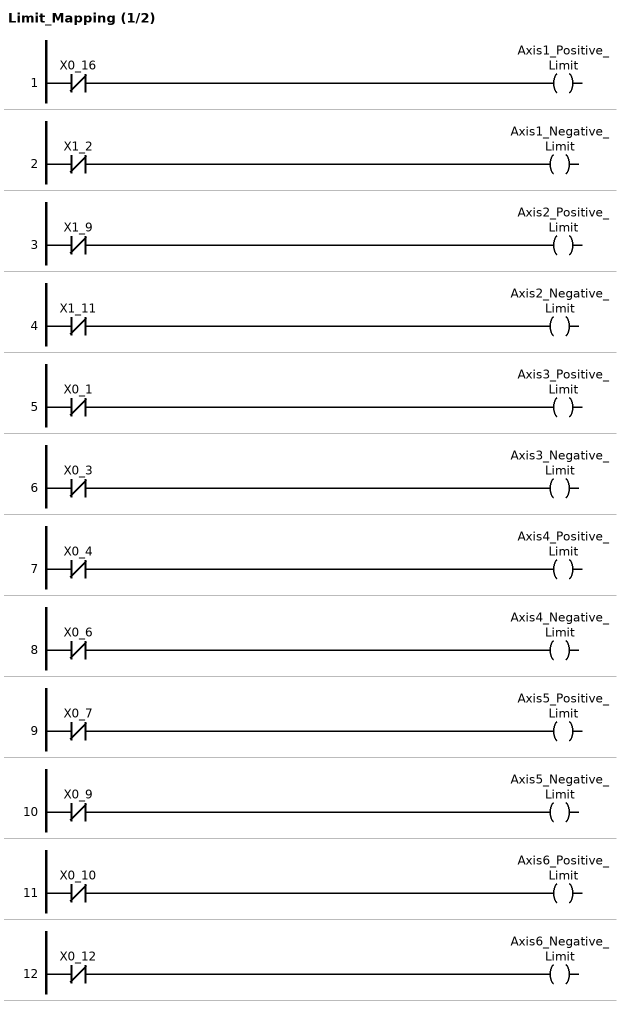
[picture p48: Limit_Mapping (LD)]
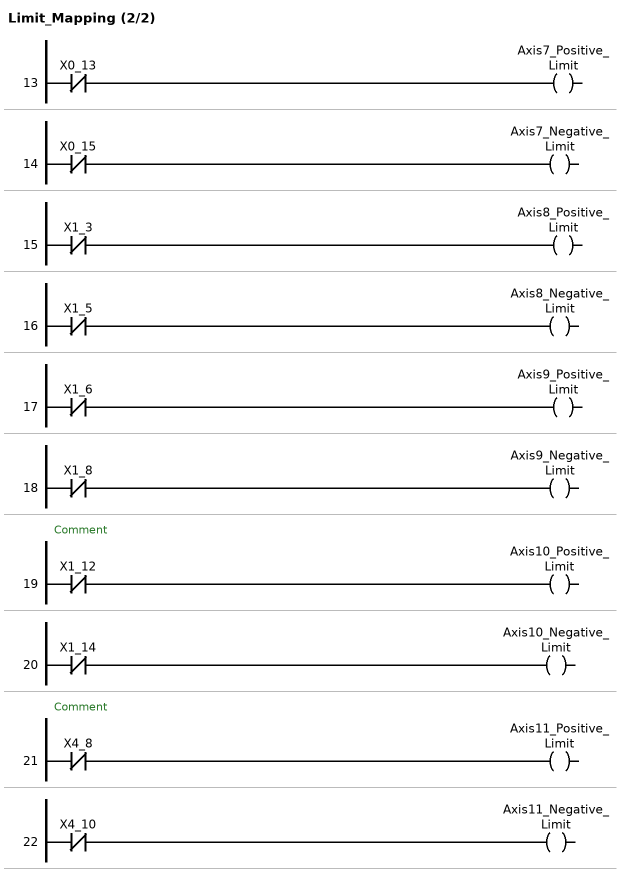
_LD_ (* Ladder Diagram *)
NETWORK 1
	[/X0_16] --- (Axis1_Positive_Limit)
NETWORK 2
	[/X1_2] --- (Axis1_Negative_Limit)
NETWORK 3
	[/X1_9] --- (Axis2_Positive_Limit)
NETWORK 4
	[/X1_11] --- (Axis2_Negative_Limit)
NETWORK 5
	[/X0_1] --- (Axis3_Positive_Limit)
NETWORK 6
	[/X0_3] --- (Axis3_Negative_Limit)
NETWORK 7
	[/X0_4] --- (Axis4_Positive_Limit)
NETWORK 8
	[/X0_6] --- (Axis4_Negative_Limit)
NETWORK 9
	[/X0_7] --- (Axis5_Positive_Limit)
NETWORK 10
	[/X0_9] --- (Axis5_Negative_Limit)
NETWORK 11
	[/X0_10] --- (Axis6_Positive_Limit)
NETWORK 12
	[/X0_12] --- (Axis6_Negative_Limit)
NETWORK 13
	[/X0_13] --- (Axis7_Positive_Limit)
NETWORK 14
	[/X0_15] --- (Axis7_Negative_Limit)
NETWORK 15
	[/X1_3] --- (Axis8_Positive_Limit)
NETWORK 16
	[/X1_5] --- (Axis8_Negative_Limit)
NETWORK 17
	[/X1_6] --- (Axis9_Positive_Limit)
NETWORK 18
	[/X1_8] --- (Axis9_Negative_Limit)
NETWORK 19 (* Comment *)
	[/X1_12] --- (Axis10_Positive_Limit)
NETWORK 20
	[/X1_14] --- (Axis10_Negative_Limit)
NETWORK 21 (* Comment *)
	[/X4_8] --- (Axis11_Positive_Limit)
NETWORK 22
	[/X4_10] --- (Axis11_Negative_Limit)
_END_LD_
(* the same logic as Structured Text *)
(* Network 1 *)
Axis1_Positive_Limit := NOT X0_16;
(* Network 2 *)
Axis1_Negative_Limit := NOT X1_2;
(* Network 3 *)
Axis2_Positive_Limit := NOT X1_9;
(* Network 4 *)
Axis2_Negative_Limit := NOT X1_11;
(* Network 5 *)
Axis3_Positive_Limit := NOT X0_1;
(* Network 6 *)
Axis3_Negative_Limit := NOT X0_3;
(* Network 7 *)
Axis4_Positive_Limit := NOT X0_4;
(* Network 8 *)
Axis4_Negative_Limit := NOT X0_6;
(* Network 9 *)
Axis5_Positive_Limit := NOT X0_7;
(* Network 10 *)
Axis5_Negative_Limit := NOT X0_9;
(* Network 11 *)
Axis6_Positive_Limit := NOT X0_10;
(* Network 12 *)
Axis6_Negative_Limit := NOT X0_12;
(* Network 13 *)
Axis7_Positive_Limit := NOT X0_13;
(* Network 14 *)
Axis7_Negative_Limit := NOT X0_15;
(* Network 15 *)
Axis8_Positive_Limit := NOT X1_3;
(* Network 16 *)
Axis8_Negative_Limit := NOT X1_5;
(* Network 17 *)
Axis9_Positive_Limit := NOT X1_6;
(* Network 18 *)
Axis9_Negative_Limit := NOT X1_8;
(* Network 19: Comment *)
Axis10_Positive_Limit := NOT X1_12;
(* Network 20 *)
Axis10_Negative_Limit := NOT X1_14;
(* Network 21: Comment *)
Axis11_Positive_Limit := NOT X4_8;
(* Network 22 *)
Axis11_Negative_Limit := NOT X4_10;
END_PROGRAM

(* POU Other_Folder/Speed_AxisStatus_IO/Speed_Setting, ST *)
PROGRAM Speed_Setting
VAR
	UP1: R_TRIG;
	UP2: R_TRIG;
	UP3: R_TRIG;

	step: INT;
END_VAR
CASE step OF
0:
step:=1;


1:
UP1(CLK:=M100 , Q=> );
UP2(CLK:=M101 , Q=> );
UP3(CLK:=M102 , Q=> );
(*调速选择*)
IF UP1.Q THEN(*低速*)
D11:=D100[0];D12:=D100[1];D13:=D100[2];D14:=D100[3];D15:=D100[4];
D16:=D100[5];D17:=D100[6];D18:=D100[7];D19:=D100[8];D20:=D100[9];D2_1:=D100[10];D2_2:=D100[11];
step:=10;
END_IF
IF UP2.Q THEN(*中速*)
D11:=D101[0];D12:=D101[1];D13:=D101[2];D14:=D101[3];D15:=D101[4];
D16:=D101[5];D17:=D101[6];D18:=D101[7];D19:=D101[8];D20:=D101[9];D2_1:=D101[10];D2_2:=D101[11];
step:=20;
END_IF
IF UP3.Q THEN(*高速*)
D11:=D102[0];D12:=D102[1];D13:=D102[2];D14:=D102[3];D15:=D102[4];
D16:=D102[5];D17:=D102[6];D18:=D102[7];D19:=D102[8];D20:=D102[9];D2_1:=D102[10];D2_2:=D102[11];
step:=30;
END_IF

10:
M101:=FALSE;
M102:=FALSE;
step:=1;

20:
M100:=FALSE;
M102:=FALSE;
step:=1;

30:
M100:=FALSE;
M101:=FALSE;
step:=1;


END_CASE
END_PROGRAM

(* POU Debug_Folder/Axis1_Debug_Model, ST *)
PROGRAM Axis1_Debug_Model
VAR
	UP1: R_TRIG;
	UP2: R_TRIG;
	UP3: R_TRIG;
	UP4: R_TRIG;
	step:INT;
END_VAR
UP1(CLK:=Axis1_debug_trigger , Q=> );

CASE step OF
0:
IF UP1.Q THEN
step:=1;
END_IF;

1:
(*点动加-----------
点动减------------
手动点动-----------*)
UP2(CLK:=Axis1_mov_add , Q=> );
UP3(CLK:=Axis1_mov_sub , Q=> );
UP4(CLK:=Axis1_mov_line , Q=> );

IF UP2.Q AND Debug_Model AND Axis1_Poweron AND NOT Total_Pause THEN
D1:=Axis1.NcToPlc.ActPos+D200;
Axis1_mov_add:=FALSE;
step:=10;
ELSE
Axis1_mov_add:=FALSE;
Axis1_MoveAbsolute:=FALSE;
END_IF

IF UP3.Q AND Debug_Model AND Axis1_Poweron AND NOT Total_Pause THEN
D1:=Axis1.NcToPlc.ActPos-D200;
Axis1_mov_sub:=FALSE;
step:=10;
ELSE
Axis1_mov_sub:=FALSE;
Axis1_MoveAbsolute:=FALSE;
END_IF

IF UP4.Q AND Debug_Model AND Axis1_Poweron  AND NOT Total_Pause THEN
D1:=D201;
Axis1_mov_line:=FALSE;
step:=10;
ELSE
Axis1_mov_line:=FALSE;
Axis1_MoveAbsolute:=FALSE;
END_IF

10:
Axis1_MoveAbsolute:=TRUE;
IF Axis1_Abs_Function.Done THEN
Axis1_MoveAbsolute:=FALSE;
step:=1;
END_IF

END_CASE

IF Axis1_mov_add THEN
Axis1_mov_add:=FALSE;
END_IF
IF Axis1_mov_sub THEN
Axis1_mov_sub:=FALSE;
END_IF
IF Axis1_mov_line THEN
Axis1_mov_line:=FALSE;
END_IF


IF NOT Debug_Model  THEN
Axis1_debug_trigger:=FALSE;
step:=0;
END_IF

IF Total_Emergency THEN
Axis1_debug_trigger:=FALSE;
Axis1_mov_add:=FALSE;
Axis1_mov_sub:=FALSE;
Axis1_mov_line:=FALSE;
Axis1_MoveAbsolute:=FALSE;
step:=0;
END_IF
END_PROGRAM

(* POU Debug_Folder/Axis2_Debug_Model, ST *)
PROGRAM Axis2_Debug_Model
VAR
	UP1: R_TRIG;
	UP2: R_TRIG;
	UP3: R_TRIG;
	UP4: R_TRIG;
	step:INT;

END_VAR
UP1(CLK:=Axis2_debug_trigger , Q=> );

CASE step OF
0:
IF UP1.Q THEN
step:=1;
END_IF;

1:
UP2(CLK:=Axis2_mov_add , Q=> );
UP3(CLK:=Axis2_mov_sub , Q=> );
UP4(CLK:=Axis2_mov_line , Q=> );

IF UP2.Q AND Debug_Model AND Axis2_Poweron AND NOT Total_Pause THEN
D2:=Axis2.NcToPlc.ActPos+D200;
Axis2_mov_add:=FALSE;
step:=10;
ELSE
Axis2_mov_add:=FALSE;
Axis2_MoveAbsolute:=FALSE;
END_IF

IF UP3.Q AND Debug_Model AND Axis2_Poweron AND NOT Total_Pause THEN
D2:=Axis2.NcToPlc.ActPos-D200;
Axis2_mov_sub:=FALSE;
step:=10;
ELSE
Axis2_mov_sub:=FALSE;
Axis2_MoveAbsolute:=FALSE;
END_IF

IF UP4.Q AND Debug_Model AND Axis2_Poweron AND NOT Total_Pause THEN
D2:=D202;
Axis2_mov_line:=FALSE;
step:=10;
ELSE
Axis2_mov_line:=FALSE;
Axis2_MoveAbsolute:=FALSE;
END_IF

10:
Axis2_MoveAbsolute:=TRUE;
IF Axis2_Abs_Function.Done THEN
Axis2_MoveAbsolute:=FALSE;
step:=1;
END_IF

END_CASE

IF Axis2_mov_add THEN
Axis2_mov_add:=FALSE;
END_IF
IF Axis2_mov_sub THEN
Axis2_mov_sub:=FALSE;
END_IF
IF Axis2_mov_line THEN
Axis2_mov_line:=FALSE;
END_IF


IF NOT Debug_Model  THEN
Axis2_debug_trigger:=FALSE;
step:=0;
END_IF

IF Total_Emergency THEN
Axis2_debug_trigger:=FALSE;
Axis2_mov_add:=FALSE;
Axis2_mov_sub:=FALSE;
Axis2_mov_line:=FALSE;
Axis2_MoveAbsolute:=FALSE;
step:=0;
END_IF
END_PROGRAM

(* POU Debug_Folder/Axis3_Debug_Model, ST *)
PROGRAM Axis3_Debug_Model
VAR
	UP1: R_TRIG;
	UP2: R_TRIG;
	UP3: R_TRIG;
	UP4: R_TRIG;
	step:INT;
END_VAR
UP1(CLK:=Axis3_debug_trigger , Q=> );

CASE step OF
0:
IF UP1.Q THEN
step:=1;
END_IF;

1:
UP2(CLK:=Axis3_mov_add , Q=> );
UP3(CLK:=Axis3_mov_sub , Q=> );
UP4(CLK:=Axis3_mov_line , Q=> );

IF UP2.Q AND Debug_Model AND Axis3_Poweron AND NOT Total_Pause THEN
D3:=Axis3.NcToPlc.ActPos+D200;
Axis3_mov_add:=FALSE;
step:=10;
ELSE
Axis3_mov_add:=FALSE;
Axis3_MoveAbsolute:=FALSE;
END_IF

IF UP3.Q AND Debug_Model AND Axis3_Poweron AND NOT Total_Pause THEN
D3:=Axis3.NcToPlc.ActPos-D200;
Axis3_mov_sub:=FALSE;
step:=10;
ELSE
Axis3_mov_sub:=FALSE;
Axis3_MoveAbsolute:=FALSE;
END_IF

IF UP4.Q AND Debug_Model AND Axis3_Poweron AND NOT Total_Pause THEN
D3:=D203;
Axis3_mov_line:=FALSE;
step:=10;
ELSE
Axis3_mov_line:=FALSE;
Axis3_MoveAbsolute:=FALSE;
END_IF

10:
Axis3_MoveAbsolute:=TRUE;
IF Axis3_Abs_Function.Done THEN
Axis3_MoveAbsolute:=FALSE;
step:=1;
END_IF

END_CASE

IF Axis3_mov_add THEN
Axis3_mov_add:=FALSE;
END_IF
IF Axis3_mov_sub THEN
Axis3_mov_sub:=FALSE;
END_IF
IF Axis3_mov_line THEN
Axis3_mov_line:=FALSE;
END_IF


IF NOT Debug_Model  THEN
Axis3_debug_trigger:=FALSE;
step:=0;
END_IF

IF Total_Emergency THEN
Axis3_debug_trigger:=FALSE;
Axis3_mov_add:=FALSE;
Axis3_mov_sub:=FALSE;
Axis3_mov_line:=FALSE;
Axis3_MoveAbsolute:=FALSE;
step:=0;
END_IF
END_PROGRAM

(* POU Debug_Folder/Axis4_Debug_Model, ST *)
PROGRAM Axis4_Debug_Model
VAR
	UP1: R_TRIG;
	UP2: R_TRIG;
	UP3: R_TRIG;
	UP4: R_TRIG;
	step:INT;
	M1:BOOL;


END_VAR
UP1(CLK:=Axis4_debug_trigger , Q=> );

CASE step OF
0:
IF UP1.Q THEN
step:=1;
END_IF;

1:
UP2(CLK:=Axis4_mov_add , Q=> );
IF UP2.Q AND Debug_Model AND Axis4_Poweron  AND NOT Total_Pause THEN
D4:=Axis4.NcToPlc.ActPos+D200;
Axis4_mov_add:=FALSE;
step:=10;
ELSE
Axis4_mov_add:=FALSE;
Axis4_MoveAbsolute:=FALSE;
END_IF


UP3(CLK:=Axis4_mov_sub , Q=> );
IF UP3.Q AND Debug_Model AND Axis4_Poweron  AND NOT Total_Pause  THEN
D4:=Axis4.NcToPlc.ActPos-D200;
Axis4_mov_sub:=FALSE;
step:=10;
ELSE
Axis4_mov_sub:=FALSE;
Axis4_MoveAbsolute:=FALSE;
END_IF


UP4(CLK:=Axis4_mov_line , Q=> );
IF UP4.Q AND Debug_Model AND Axis4_Poweron  AND NOT Total_Pause  THEN
D4:=D204;
Axis4_mov_line:=FALSE;
step:=10;
ELSE
Axis4_mov_line:=FALSE;
Axis4_MoveAbsolute:=FALSE;
END_IF


10:
Axis4_MoveAbsolute:=TRUE;
IF Axis4_Abs_Function.Done THEN
Axis4_MoveAbsolute:=FALSE;
step:=1;
END_IF


END_CASE

IF Axis4_mov_add THEN
Axis4_mov_add:=FALSE;
END_IF
IF Axis4_mov_sub THEN
Axis4_mov_sub:=FALSE;
END_IF
IF Axis4_mov_line THEN
Axis4_mov_line:=FALSE;
END_IF


IF NOT Debug_Model  THEN
Axis4_debug_trigger:=FALSE;
step:=0;
END_IF

IF Total_Emergency THEN
Axis4_debug_trigger:=FALSE;
Axis4_mov_add:=FALSE;
Axis4_mov_sub:=FALSE;
Axis4_mov_line:=FALSE;
Axis4_MoveAbsolute:=FALSE;
Axis4_1_MoveAbsolute:=FALSE;
step:=0;
END_IF
END_PROGRAM

(* POU Debug_Folder/Axis5_Debug_Model, ST *)
PROGRAM Axis5_Debug_Model
VAR
	UP1: R_TRIG;
	UP2: R_TRIG;
	UP3: R_TRIG;
	UP4: R_TRIG;
	step:INT;
END_VAR
UP1(CLK:=Axis5_debug_trigger , Q=> );

CASE step OF
0:
IF UP1.Q THEN
step:=1;
END_IF;

1:
UP2(CLK:=Axis5_mov_add , Q=> );
UP3(CLK:=Axis5_mov_sub , Q=> );
UP4(CLK:=Axis5_mov_line , Q=> );

IF UP2.Q AND Debug_Model AND Axis5_Poweron  AND NOT Total_Pause THEN
D5:=Axis5.NcToPlc.ActPos+D200;
Axis5_mov_add:=FALSE;
step:=10;
ELSE
Axis5_mov_add:=FALSE;
Axis5_MoveAbsolute:=FALSE;
END_IF

IF UP3.Q AND Debug_Model AND Axis5_Poweron AND NOT Total_Pause THEN
D5:=Axis5.NcToPlc.ActPos-D200;
Axis5_mov_sub:=FALSE;
step:=10;
ELSE
Axis5_mov_sub:=FALSE;
Axis5_MoveAbsolute:=FALSE;
END_IF

IF UP4.Q AND Debug_Model AND Axis5_Poweron  AND NOT Total_Pause THEN
D5:=D205;
Axis5_mov_line:=FALSE;
step:=10;
ELSE
Axis5_mov_line:=FALSE;
Axis5_MoveAbsolute:=FALSE;
END_IF

10:
Axis5_MoveAbsolute:=TRUE;
IF Axis5_Abs_Function.Done THEN
Axis5_MoveAbsolute:=FALSE;
step:=1;
END_IF

END_CASE

IF Axis5_mov_add THEN
Axis5_mov_add:=FALSE;
END_IF
IF Axis5_mov_sub THEN
Axis5_mov_sub:=FALSE;
END_IF
IF Axis5_mov_line THEN
Axis5_mov_line:=FALSE;
END_IF


IF NOT Debug_Model  THEN
Axis5_debug_trigger:=FALSE;
step:=0;
END_IF

IF Total_Emergency THEN
Axis5_debug_trigger:=FALSE;
Axis5_mov_add:=FALSE;
Axis5_mov_sub:=FALSE;
Axis5_mov_line:=FALSE;
Axis5_MoveAbsolute:=FALSE;
Axis5_1_MoveAbsolute:=FALSE;
step:=0;
END_IF
END_PROGRAM

(* POU Debug_Folder/Axis6_Debug_Model, ST *)
PROGRAM Axis6_Debug_Model
VAR
	UP1: R_TRIG;
	UP2: R_TRIG;
	UP3: R_TRIG;
	UP4: R_TRIG;
	step:INT;
END_VAR
UP1(CLK:=Axis6_debug_trigger , Q=> );

CASE step OF
0:
IF UP1.Q THEN
step:=1;
END_IF;

1:
UP2(CLK:=Axis6_mov_add , Q=> );
UP3(CLK:=Axis6_mov_sub , Q=> );
UP4(CLK:=Axis6_mov_line , Q=> );

IF UP2.Q AND Debug_Model AND Axis6_Poweron  AND NOT Total_Pause THEN
D6:=Axis6.NcToPlc.ActPos+D200;
Axis6_mov_add:=FALSE;
step:=10;
ELSE
Axis6_mov_add:=FALSE;
Axis6_MoveAbsolute:=FALSE;
END_IF

IF UP3.Q AND Debug_Model AND Axis6_Poweron AND NOT Total_Pause THEN
D6:=Axis6.NcToPlc.ActPos-D200;
Axis6_mov_sub:=FALSE;
step:=10;
ELSE
Axis6_mov_sub:=FALSE;
Axis6_MoveAbsolute:=FALSE;
END_IF

IF UP4.Q AND Debug_Model AND Axis6_Poweron  AND NOT Total_Pause THEN
D6:=D206;
Axis6_mov_line:=FALSE;
step:=10;
ELSE
Axis6_mov_line:=FALSE;
Axis6_MoveAbsolute:=FALSE;
END_IF

10:
Axis6_MoveAbsolute:=TRUE;
IF Axis6_Abs_Function.Done THEN
Axis6_MoveAbsolute:=FALSE;
step:=1;
END_IF
END_CASE

IF Axis6_mov_add THEN
Axis6_mov_add:=FALSE;
END_IF
IF Axis6_mov_sub THEN
Axis6_mov_sub:=FALSE;
END_IF
IF Axis6_mov_line THEN
Axis6_mov_line:=FALSE;
END_IF


IF NOT Debug_Model  THEN
Axis6_debug_trigger:=FALSE;
step:=0;
END_IF

IF Total_Emergency THEN
Axis6_debug_trigger:=FALSE;
Axis6_mov_add:=FALSE;
Axis6_mov_sub:=FALSE;
Axis6_mov_line:=FALSE;
Axis6_MoveAbsolute:=FALSE;
step:=0;
END_IF
END_PROGRAM

(* POU Debug_Folder/Axis7_Debug_Model, ST *)
PROGRAM Axis7_Debug_Model
VAR
	UP1: R_TRIG;
	UP2: R_TRIG;
	UP3: R_TRIG;
	UP4: R_TRIG;
	step:INT;
END_VAR
UP1(CLK:=Axis7_debug_trigger , Q=> );

CASE step OF
0:
IF UP1.Q THEN
step:=1;
END_IF;

1:
UP2(CLK:=Axis7_mov_add , Q=> );
UP3(CLK:=Axis7_mov_sub , Q=> );
UP4(CLK:=Axis7_mov_line , Q=> );

IF UP2.Q AND Debug_Model AND Axis7_Poweron  AND NOT Total_Pause THEN
D7:=Axis7.NcToPlc.ActPos+D200;
Axis7_mov_add:=FALSE;
step:=10;
ELSE
Axis7_mov_add:=FALSE;
Axis7_MoveAbsolute:=FALSE;
END_IF

IF UP3.Q AND Debug_Model AND Axis7_Poweron AND NOT Total_Pause THEN
D7:=Axis7.NcToPlc.ActPos-D200;
Axis7_mov_sub:=FALSE;
step:=10;
ELSE
Axis7_mov_sub:=FALSE;
Axis7_MoveAbsolute:=FALSE;
END_IF

IF UP4.Q AND Debug_Model AND Axis7_Poweron  AND NOT Total_Pause THEN
D7:=D207;
Axis7_mov_line:=FALSE;
step:=10;
ELSE
Axis7_mov_line:=FALSE;
Axis7_MoveAbsolute:=FALSE;
END_IF

10:
Axis7_MoveAbsolute:=TRUE;
IF Axis7_Abs_Function.Done THEN
Axis7_MoveAbsolute:=FALSE;
step:=1;
END_IF
END_CASE

IF Axis7_mov_add THEN
Axis7_mov_add:=FALSE;
END_IF
IF Axis7_mov_sub THEN
Axis7_mov_sub:=FALSE;
END_IF
IF Axis7_mov_line THEN
Axis7_mov_line:=FALSE;
END_IF


IF NOT Debug_Model  THEN
Axis7_debug_trigger:=FALSE;
step:=0;
END_IF

IF Total_Emergency THEN
Axis7_debug_trigger:=FALSE;
Axis7_mov_add:=FALSE;
Axis7_mov_sub:=FALSE;
Axis7_mov_line:=FALSE;
Axis7_MoveAbsolute:=FALSE;
step:=0;
END_IF
END_PROGRAM

(* POU Debug_Folder/Axis8_Debug_Model, ST *)
PROGRAM Axis8_Debug_Model
VAR
	UP1: R_TRIG;
	UP2: R_TRIG;
	UP3: R_TRIG;
	UP4: R_TRIG;
	step:INT;
END_VAR
UP1(CLK:=Axis8_debug_trigger , Q=> );

CASE step OF
0:
IF UP1.Q THEN
step:=1;
END_IF;

1:
UP2(CLK:=Axis8_mov_add , Q=> );
UP3(CLK:=Axis8_mov_sub , Q=> );
UP4(CLK:=Axis8_mov_line , Q=> );

IF UP2.Q AND Debug_Model AND Axis8_Poweron  AND NOT Total_Pause THEN
D8:=Axis8.NcToPlc.ActPos+D200;
Axis8_mov_add:=FALSE;
step:=10;
ELSE
Axis8_mov_add:=FALSE;
Axis8_MoveAbsolute:=FALSE;
END_IF

IF UP3.Q AND Debug_Model AND Axis8_Poweron AND NOT Total_Pause THEN
D8:=Axis8.NcToPlc.ActPos-D200;
Axis8_mov_sub:=FALSE;
step:=10;
ELSE
Axis8_mov_sub:=FALSE;
Axis8_MoveAbsolute:=FALSE;
END_IF

IF UP4.Q AND Debug_Model AND Axis8_Poweron  AND NOT Total_Pause THEN
D8:=D208;
Axis8_mov_line:=FALSE;
step:=10;
ELSE
Axis8_mov_line:=FALSE;
Axis8_MoveAbsolute:=FALSE;
END_IF

10:
Axis8_MoveAbsolute:=TRUE;
IF Axis8_Abs_Function.Done THEN
Axis8_MoveAbsolute:=FALSE;
step:=1;
END_IF
END_CASE

IF Axis8_mov_add THEN
Axis8_mov_add:=FALSE;
END_IF
IF Axis8_mov_sub THEN
Axis8_mov_sub:=FALSE;
END_IF
IF Axis8_mov_line THEN
Axis8_mov_line:=FALSE;
END_IF


IF NOT Debug_Model  THEN
Axis8_debug_trigger:=FALSE;
step:=0;
END_IF

IF Total_Emergency THEN
Axis8_debug_trigger:=FALSE;
Axis8_mov_add:=FALSE;
Axis8_mov_sub:=FALSE;
Axis8_mov_line:=FALSE;
Axis8_MoveAbsolute:=FALSE;
step:=0;
END_IF
END_PROGRAM

(* POU Debug_Folder/Axis9_Debug_Model, ST *)
PROGRAM Axis9_Debug_Model
VAR
	UP1: R_TRIG;
	UP2: R_TRIG;
	UP3: R_TRIG;
	UP4: R_TRIG;
	step:INT;
END_VAR
UP1(CLK:=Axis9_debug_trigger , Q=> );

CASE step OF
0:
IF UP1.Q THEN
step:=1;
END_IF;

1:
UP2(CLK:=Axis9_mov_add , Q=> );
UP3(CLK:=Axis9_mov_sub , Q=> );
UP4(CLK:=Axis9_mov_line , Q=> );

IF UP2.Q AND Debug_Model AND Axis9_Poweron  AND NOT Total_Pause THEN
D9:=Axis9.NcToPlc.ActPos+D200;
Axis9_mov_add:=FALSE;
step:=10;
ELSE
Axis9_mov_add:=FALSE;
Axis9_MoveAbsolute:=FALSE;
END_IF

IF UP3.Q AND Debug_Model AND Axis9_Poweron AND NOT Total_Pause THEN
D9:=Axis9.NcToPlc.ActPos-D200;
Axis9_mov_sub:=FALSE;
step:=10;
ELSE
Axis9_mov_sub:=FALSE;
Axis9_MoveAbsolute:=FALSE;
END_IF

IF UP4.Q AND Debug_Model AND Axis9_Poweron  AND NOT Total_Pause THEN
D9:=D209;
Axis9_mov_line:=FALSE;
step:=10;
ELSE
Axis9_mov_line:=FALSE;
Axis9_MoveAbsolute:=FALSE;
END_IF

10:
Axis9_MoveAbsolute:=TRUE;
IF Axis9_Abs_Function.Done THEN
Axis9_MoveAbsolute:=FALSE;
step:=1;
END_IF
END_CASE

IF Axis9_mov_add THEN
Axis9_mov_add:=FALSE;
END_IF
IF Axis9_mov_sub THEN
Axis9_mov_sub:=FALSE;
END_IF
IF Axis9_mov_line THEN
Axis9_mov_line:=FALSE;
END_IF


IF NOT Debug_Model  THEN
Axis9_debug_trigger:=FALSE;
step:=0;
END_IF

IF Total_Emergency THEN
Axis9_debug_trigger:=FALSE;
Axis9_mov_add:=FALSE;
Axis9_mov_sub:=FALSE;
Axis9_mov_line:=FALSE;
Axis9_MoveAbsolute:=FALSE;
step:=0;
END_IF
END_PROGRAM

(* POU Debug_Folder/Axis10_Debug_Model, ST *)
PROGRAM Axis10_Debug_Model
VAR
	UP1: R_TRIG;
	UP2: R_TRIG;
	UP3: R_TRIG;
	UP4: R_TRIG;
	step:INT;
END_VAR
UP1(CLK:=Axis10_debug_trigger , Q=> );

CASE step OF
0:
IF UP1.Q THEN
step:=1;
END_IF;

1:
UP2(CLK:=Axis10_mov_add , Q=> );
UP3(CLK:=Axis10_mov_sub , Q=> );
UP4(CLK:=Axis10_mov_line , Q=> );

IF UP2.Q AND Debug_Model AND Axis10_Poweron  AND NOT Total_Pause THEN
D10:=Axis10.NcToPlc.ActPos+D200;
Axis10_mov_add:=FALSE;
step:=10;
ELSE
Axis10_mov_add:=FALSE;
Axis10_MoveAbsolute:=FALSE;
END_IF

IF UP3.Q AND Debug_Model AND Axis10_Poweron AND NOT Total_Pause THEN
D10:=Axis10.NcToPlc.ActPos-D200;
Axis10_mov_sub:=FALSE;
step:=10;
ELSE
Axis10_mov_sub:=FALSE;
Axis10_MoveAbsolute:=FALSE;
END_IF

IF UP4.Q AND Debug_Model AND Axis10_Poweron  AND NOT Total_Pause THEN
D10:=D210;
Axis10_mov_line:=FALSE;
step:=10;
ELSE
Axis10_mov_line:=FALSE;
Axis10_MoveAbsolute:=FALSE;
END_IF

10:
Axis10_MoveAbsolute:=TRUE;
IF Axis10_Abs_Function.Done THEN
Axis10_MoveAbsolute:=FALSE;
step:=1;
END_IF
END_CASE

IF Axis10_mov_add THEN
Axis10_mov_add:=FALSE;
END_IF
IF Axis10_mov_sub THEN
Axis10_mov_sub:=FALSE;
END_IF
IF Axis10_mov_line THEN
Axis10_mov_line:=FALSE;
END_IF


IF NOT Debug_Model  THEN
Axis10_debug_trigger:=FALSE;
step:=0;
END_IF

IF Total_Emergency THEN
Axis10_debug_trigger:=FALSE;
Axis10_mov_add:=FALSE;
Axis10_mov_sub:=FALSE;
Axis10_mov_line:=FALSE;
Axis10_MoveAbsolute:=FALSE;
step:=0;
END_IF
END_PROGRAM

(* POU Debug_Folder/Axis11_Debug_Model, ST *)
PROGRAM Axis11_Debug_Model
VAR

	UP1: R_TRIG;
	UP2: R_TRIG;
	UP3: R_TRIG;
	UP4: R_TRIG;
	step:INT;
END_VAR
UP1(CLK:=Axis11_debug_trigger , Q=> );

CASE step OF
0:
IF UP1.Q THEN
step:=1;
END_IF;

1:
UP2(CLK:=Axis11_mov_add , Q=> );
UP3(CLK:=Axis11_mov_sub , Q=> );
UP4(CLK:=Axis11_mov_line , Q=> );

IF UP2.Q AND Debug_Model AND Axis11_Poweron  AND NOT Total_Pause THEN
D1_1:=Axis11.NcToPlc.ActPos+D200;
Axis11_mov_add:=FALSE;
step:=10;
ELSE
Axis11_mov_add:=FALSE;
Axis11_MoveAbsolute:=FALSE;
END_IF

IF UP3.Q AND Debug_Model AND Axis11_Poweron AND NOT Total_Pause THEN
D1_1:=Axis11.NcToPlc.ActPos-D200;
Axis11_mov_sub:=FALSE;
step:=10;
ELSE
Axis11_mov_sub:=FALSE;
Axis11_MoveAbsolute:=FALSE;
END_IF

IF UP4.Q AND Debug_Model AND Axis11_Poweron  AND NOT Total_Pause THEN
D1_1:=D211;
Axis11_mov_line:=FALSE;
step:=10;
ELSE
Axis11_mov_line:=FALSE;
Axis11_MoveAbsolute:=FALSE;
END_IF

10:
Axis11_MoveAbsolute:=TRUE;
IF Axis11_Abs_Function.Done THEN
Axis11_MoveAbsolute:=FALSE;
step:=1;
END_IF
END_CASE

IF Axis11_mov_add THEN
Axis11_mov_add:=FALSE;
END_IF
IF Axis11_mov_sub THEN
Axis11_mov_sub:=FALSE;
END_IF
IF Axis11_mov_line THEN
Axis11_mov_line:=FALSE;
END_IF


IF NOT Debug_Model  THEN
Axis11_debug_trigger:=FALSE;
step:=0;
END_IF

IF Total_Emergency THEN
Axis11_debug_trigger:=FALSE;
Axis11_mov_add:=FALSE;
Axis11_mov_sub:=FALSE;
Axis11_mov_line:=FALSE;
Axis11_MoveAbsolute:=FALSE;
step:=0;
END_IF
END_PROGRAM

(* POU Debug_Folder/Others_Debug_Model, LD *)
PROGRAM Others_Debug_Model
VAR
END_VAR
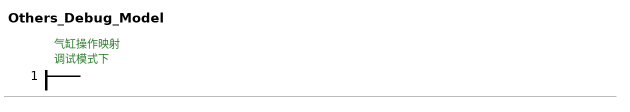
_LD_ (* Ladder Diagram *)
NETWORK 1 (* 气缸操作映射 / 调试模式下 *)
	*
_END_LD_
(* the same logic as Structured Text *)
(* Network 1: 气缸操作映射 / 调试模式下 *)
END_PROGRAM

(* POU Other_Folder/Akam_Stop_Message/Initialization_Folder/Debug12, LD *)
	PROGRAM Debug12
VAR
	t1: TON;
END_VAR
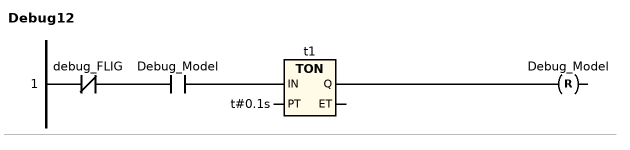
_LD_ (* Ladder Diagram *)
NETWORK 1
	[/debug_FLIG] - [Debug_Model] - t1:TON(IN: *, PT: t#0.1s) --- (R Debug_Model)
_END_LD_
(* the same logic as Structured Text *)
(* Network 1 *)
t1(IN := NOT debug_FLIG AND Debug_Model, PT := t#0.1s);
IF t1.Q THEN Debug_Model := FALSE; END_IF;
END_PROGRAM

(* POU Run_Main_Folder/Feed_alam_status, LD *)
PROGRAM Feed_alam_status
VAR


END_VAR
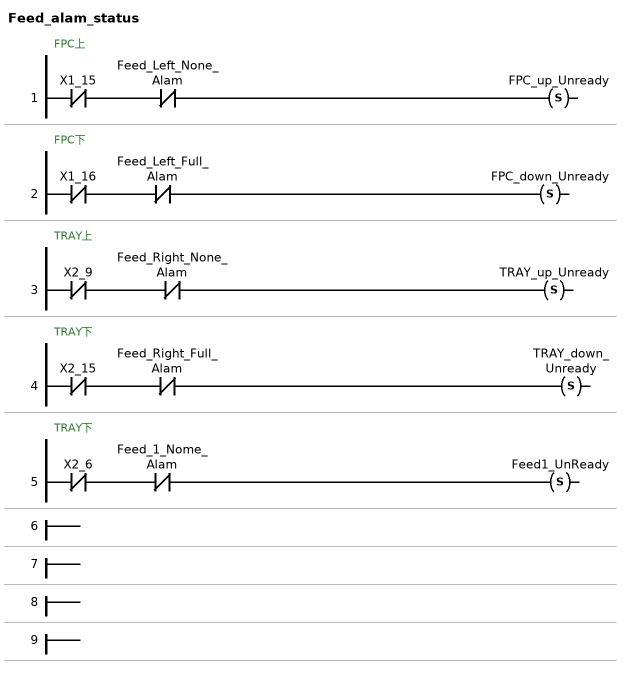
_LD_ (* Ladder Diagram *)
NETWORK 1 (* FPC上 *)
	[/X1_15] - [/Feed_Left_None_Alam] --- (S FPC_up_Unready)
NETWORK 2 (* FPC下 *)
	[/X1_16] - [/Feed_Left_Full_Alam] --- (S FPC_down_Unready)
NETWORK 3 (* TRAY上 *)
	[/X2_9] - [/Feed_Right_None_Alam] --- (S TRAY_up_Unready)
NETWORK 4 (* TRAY下 *)
	[/X2_15] - [/Feed_Right_Full_Alam] --- (S TRAY_down_Unready)
NETWORK 5 (* TRAY下 *)
	[/X2_6] - [/Feed_1_Nome_Alam] --- (S Feed1_UnReady)
NETWORK 6
	*
NETWORK 7
	*
NETWORK 8
	*
NETWORK 9
	*
_END_LD_
(* the same logic as Structured Text *)
(* Network 1: FPC上 *)
IF NOT X1_15 AND NOT Feed_Left_None_Alam THEN FPC_up_Unready := TRUE; END_IF;
(* Network 2: FPC下 *)
IF NOT X1_16 AND NOT Feed_Left_Full_Alam THEN FPC_down_Unready := TRUE; END_IF;
(* Network 3: TRAY上 *)
IF NOT X2_9 AND NOT Feed_Right_None_Alam THEN TRAY_up_Unready := TRUE; END_IF;
(* Network 4: TRAY下 *)
IF NOT X2_15 AND NOT Feed_Right_Full_Alam THEN TRAY_down_Unready := TRUE; END_IF;
(* Network 5: TRAY下 *)
IF NOT X2_6 AND NOT Feed_1_Nome_Alam THEN Feed1_UnReady := TRUE; END_IF;
(* Network 6 *)
(* Network 7 *)
(* Network 8 *)
(* Network 9 *)
END_PROGRAM

(* POU Other_Folder/Home_Back/Axis1_Home_Back, LD *)
PROGRAM Axis1_Home_Back
VAR
	UP1: R_TRIG;
	M1: BOOL;
	M2: BOOL;
	UP2: R_TRIG;
	T1: TON;
	M3: BOOL;
	M4: BOOL;
	DOWN1: F_TRIG;
	M20: BOOL;
END_VAR
VAR (* helpers for the ST form of the networks *)
	_p1 : BOOL;
	_p2 : BOOL;
	_p3 : BOOL;
END_VAR
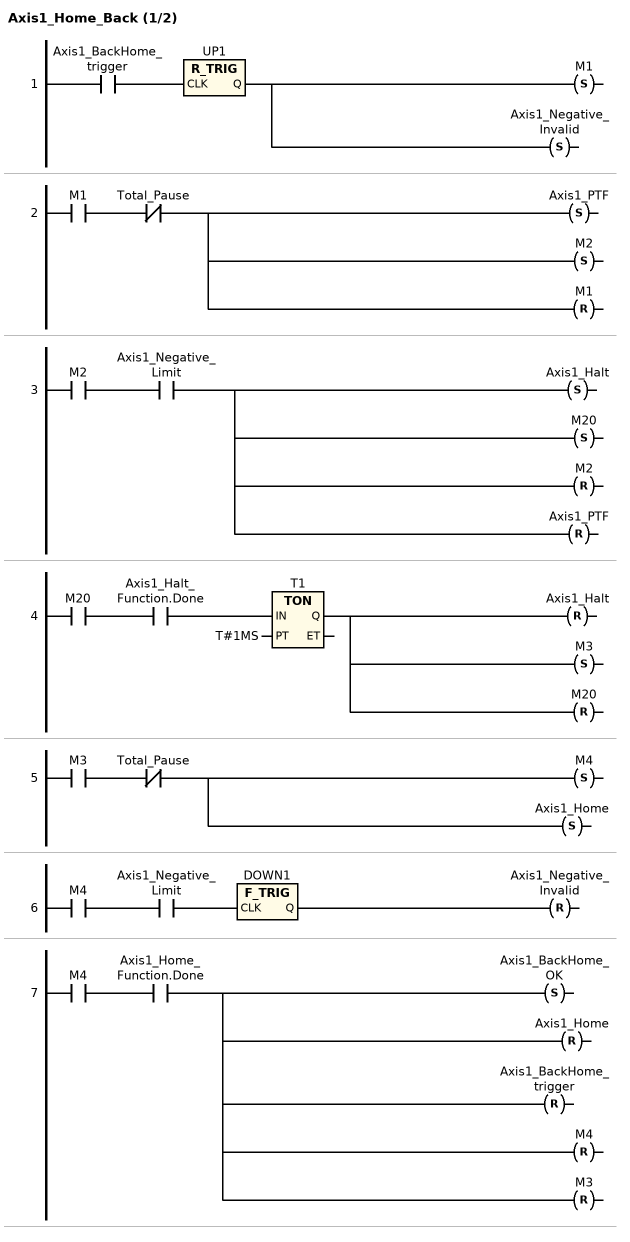
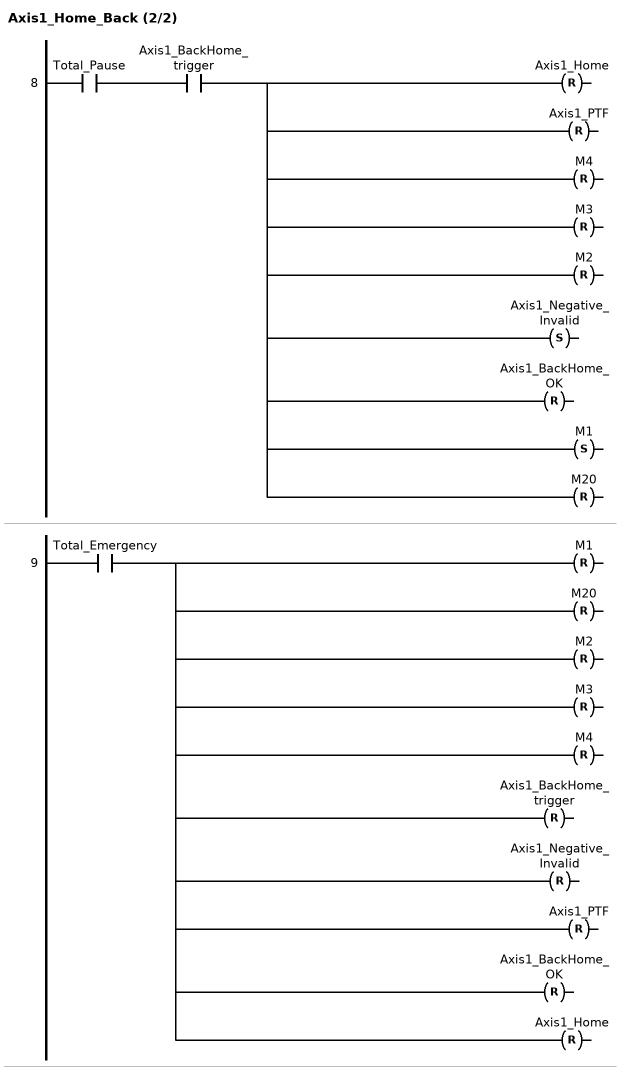
_LD_ (* Ladder Diagram *)
NETWORK 1
	[Axis1_BackHome_trigger] - UP1:R_TRIG(CLK: *) --- (S M1) (S Axis1_Negative_Invalid)
NETWORK 2
	[M1] - [/Total_Pause] --- (S Axis1_PTF) (S M2) (R M1)
NETWORK 3
	[M2] - [Axis1_Negative_Limit] --- (S Axis1_Halt) (S M20) (R M2) (R Axis1_PTF)
NETWORK 4
	[M20] - [Axis1_Halt_Function.Done] - T1:TON(IN: *, PT: T#1MS) --- (R Axis1_Halt) (S M3) (R M20)
NETWORK 5
	[M3] - [/Total_Pause] --- (S M4) (S Axis1_Home)
NETWORK 6
	[M4] - [Axis1_Negative_Limit] - DOWN1:F_TRIG(CLK: *) --- (R Axis1_Negative_Invalid)
NETWORK 7
	[M4] - [Axis1_Home_Function.Done] --- (S Axis1_BackHome_OK) (R Axis1_Home) (R Axis1_BackHome_trigger) (R M4) (R M3)
NETWORK 8
	[Total_Pause] - [Axis1_BackHome_trigger] --- (R Axis1_Home) (R Axis1_PTF) (R M4) (R M3) (R M2) (S Axis1_Negative_Invalid) (R Axis1_BackHome_OK) (S M1) (R M20)
NETWORK 9
	[Total_Emergency] --- (R M1) (R M20) (R M2) (R M3) (R M4) (R Axis1_BackHome_trigger) (R Axis1_Negative_Invalid) (R Axis1_PTF) (R Axis1_BackHome_OK) (R Axis1_Home)
_END_LD_
(* the same logic as Structured Text *)
(* Network 1 *)
UP1(CLK := Axis1_BackHome_trigger);
IF UP1.Q THEN M1 := TRUE; Axis1_Negative_Invalid := TRUE; END_IF;
(* Network 2 *)
_p1 := M1 AND NOT Total_Pause;
IF _p1 THEN Axis1_PTF := TRUE; M2 := TRUE; M1 := FALSE; END_IF;
(* Network 3 *)
_p2 := M2 AND Axis1_Negative_Limit;
IF _p2 THEN Axis1_Halt := TRUE; M20 := TRUE; M2 := FALSE; Axis1_PTF := FALSE; END_IF;
(* Network 4 *)
T1(IN := M20 AND Axis1_Halt_Function.Done, PT := T#1MS);
IF T1.Q THEN Axis1_Halt := FALSE; M3 := TRUE; M20 := FALSE; END_IF;
(* Network 5 *)
IF M3 AND NOT Total_Pause THEN M4 := TRUE; Axis1_Home := TRUE; END_IF;
(* Network 6 *)
DOWN1(CLK := M4 AND Axis1_Negative_Limit);
IF DOWN1.Q THEN Axis1_Negative_Invalid := FALSE; END_IF;
(* Network 7 *)
_p3 := M4 AND Axis1_Home_Function.Done;
IF _p3 THEN Axis1_BackHome_OK := TRUE; Axis1_Home := FALSE; Axis1_BackHome_trigger := FALSE; M4 := FALSE; M3 := FALSE; END_IF;
(* Network 8 *)
IF Total_Pause AND Axis1_BackHome_trigger THEN Axis1_Home := FALSE; Axis1_PTF := FALSE; M4 := FALSE; M3 := FALSE; M2 := FALSE; Axis1_Negative_Invalid := TRUE; Axis1_BackHome_OK := FALSE; M1 := TRUE; M20 := FALSE; END_IF;
(* Network 9 *)
IF Total_Emergency THEN M1 := FALSE; M20 := FALSE; M2 := FALSE; M3 := FALSE; M4 := FALSE; Axis1_BackHome_trigger := FALSE; Axis1_Negative_Invalid := FALSE; Axis1_PTF := FALSE; Axis1_BackHome_OK := FALSE; Axis1_Home := FALSE; END_IF;
END_PROGRAM

(* POU Other_Folder/Home_Back/Axis2_Home_Back, LD *)
PROGRAM Axis2_Home_Back
VAR
	UP1: R_TRIG;
	M1: BOOL;
	M2: BOOL;
	UP2: R_TRIG;
	T1: TON;
	M3: BOOL;
	M4: BOOL;
	DOWN1: F_TRIG;
	M20: BOOL;
END_VAR
VAR (* helpers for the ST form of the networks *)
	_p1 : BOOL;
	_p2 : BOOL;
	_p3 : BOOL;
END_VAR
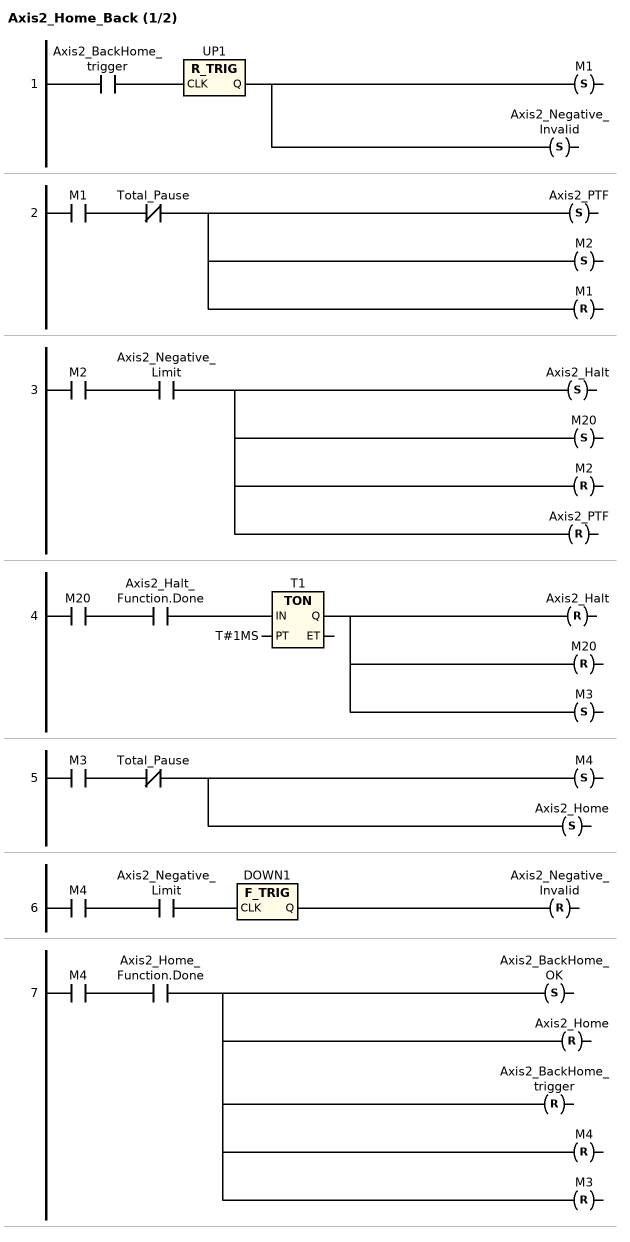
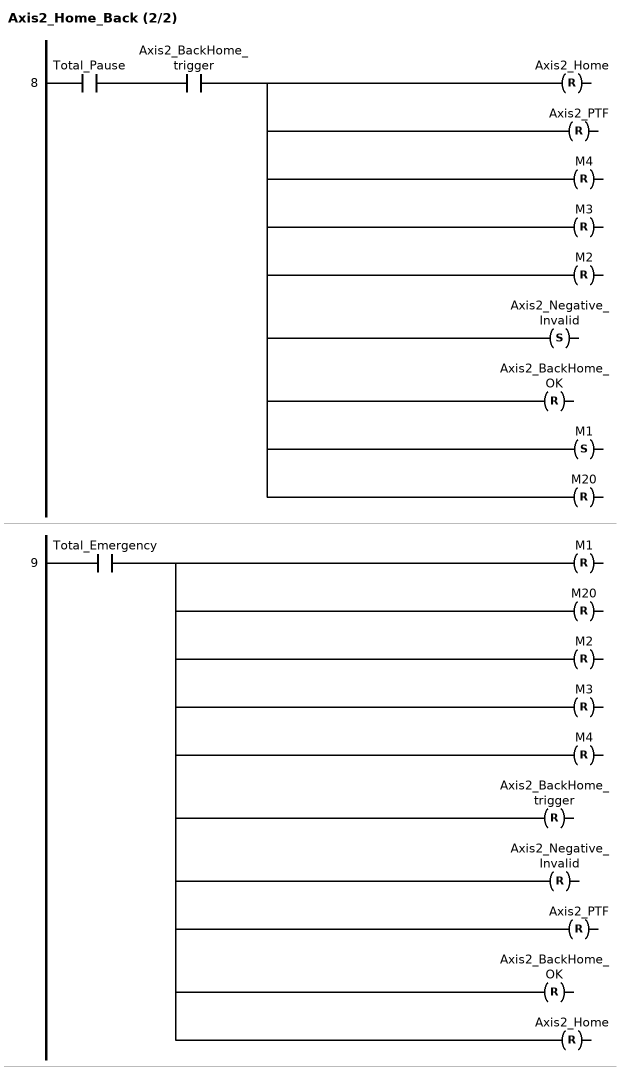
_LD_ (* Ladder Diagram *)
NETWORK 1
	[Axis2_BackHome_trigger] - UP1:R_TRIG(CLK: *) --- (S M1) (S Axis2_Negative_Invalid)
NETWORK 2
	[M1] - [/Total_Pause] --- (S Axis2_PTF) (S M2) (R M1)
NETWORK 3
	[M2] - [Axis2_Negative_Limit] --- (S Axis2_Halt) (S M20) (R M2) (R Axis2_PTF)
NETWORK 4
	[M20] - [Axis2_Halt_Function.Done] - T1:TON(IN: *, PT: T#1MS) --- (R Axis2_Halt) (R M20) (S M3)
NETWORK 5
	[M3] - [/Total_Pause] --- (S M4) (S Axis2_Home)
NETWORK 6
	[M4] - [Axis2_Negative_Limit] - DOWN1:F_TRIG(CLK: *) --- (R Axis2_Negative_Invalid)
NETWORK 7
	[M4] - [Axis2_Home_Function.Done] --- (S Axis2_BackHome_OK) (R Axis2_Home) (R Axis2_BackHome_trigger) (R M4) (R M3)
NETWORK 8
	[Total_Pause] - [Axis2_BackHome_trigger] --- (R Axis2_Home) (R Axis2_PTF) (R M4) (R M3) (R M2) (S Axis2_Negative_Invalid) (R Axis2_BackHome_OK) (S M1) (R M20)
NETWORK 9
	[Total_Emergency] --- (R M1) (R M20) (R M2) (R M3) (R M4) (R Axis2_BackHome_trigger) (R Axis2_Negative_Invalid) (R Axis2_PTF) (R Axis2_BackHome_OK) (R Axis2_Home)
_END_LD_
(* the same logic as Structured Text *)
(* Network 1 *)
UP1(CLK := Axis2_BackHome_trigger);
IF UP1.Q THEN M1 := TRUE; Axis2_Negative_Invalid := TRUE; END_IF;
(* Network 2 *)
_p1 := M1 AND NOT Total_Pause;
IF _p1 THEN Axis2_PTF := TRUE; M2 := TRUE; M1 := FALSE; END_IF;
(* Network 3 *)
_p2 := M2 AND Axis2_Negative_Limit;
IF _p2 THEN Axis2_Halt := TRUE; M20 := TRUE; M2 := FALSE; Axis2_PTF := FALSE; END_IF;
(* Network 4 *)
T1(IN := M20 AND Axis2_Halt_Function.Done, PT := T#1MS);
IF T1.Q THEN Axis2_Halt := FALSE; M20 := FALSE; M3 := TRUE; END_IF;
(* Network 5 *)
IF M3 AND NOT Total_Pause THEN M4 := TRUE; Axis2_Home := TRUE; END_IF;
(* Network 6 *)
DOWN1(CLK := M4 AND Axis2_Negative_Limit);
IF DOWN1.Q THEN Axis2_Negative_Invalid := FALSE; END_IF;
(* Network 7 *)
_p3 := M4 AND Axis2_Home_Function.Done;
IF _p3 THEN Axis2_BackHome_OK := TRUE; Axis2_Home := FALSE; Axis2_BackHome_trigger := FALSE; M4 := FALSE; M3 := FALSE; END_IF;
(* Network 8 *)
IF Total_Pause AND Axis2_BackHome_trigger THEN Axis2_Home := FALSE; Axis2_PTF := FALSE; M4 := FALSE; M3 := FALSE; M2 := FALSE; Axis2_Negative_Invalid := TRUE; Axis2_BackHome_OK := FALSE; M1 := TRUE; M20 := FALSE; END_IF;
(* Network 9 *)
IF Total_Emergency THEN M1 := FALSE; M20 := FALSE; M2 := FALSE; M3 := FALSE; M4 := FALSE; Axis2_BackHome_trigger := FALSE; Axis2_Negative_Invalid := FALSE; Axis2_PTF := FALSE; Axis2_BackHome_OK := FALSE; Axis2_Home := FALSE; END_IF;
END_PROGRAM

(* POU Other_Folder/Home_Back/Axis3_Home_Back, LD *)
PROGRAM Axis3_Home_Back
VAR
	UP1: R_TRIG;
	M1: BOOL;
	M2: BOOL;
	UP2: R_TRIG;
	T1: TON;
	M3: BOOL;
	M4: BOOL;
	DOWN1: F_TRIG;
	M20: BOOL;
END_VAR
VAR (* helpers for the ST form of the networks *)
	_p1 : BOOL;
	_p2 : BOOL;
	_p3 : BOOL;
END_VAR
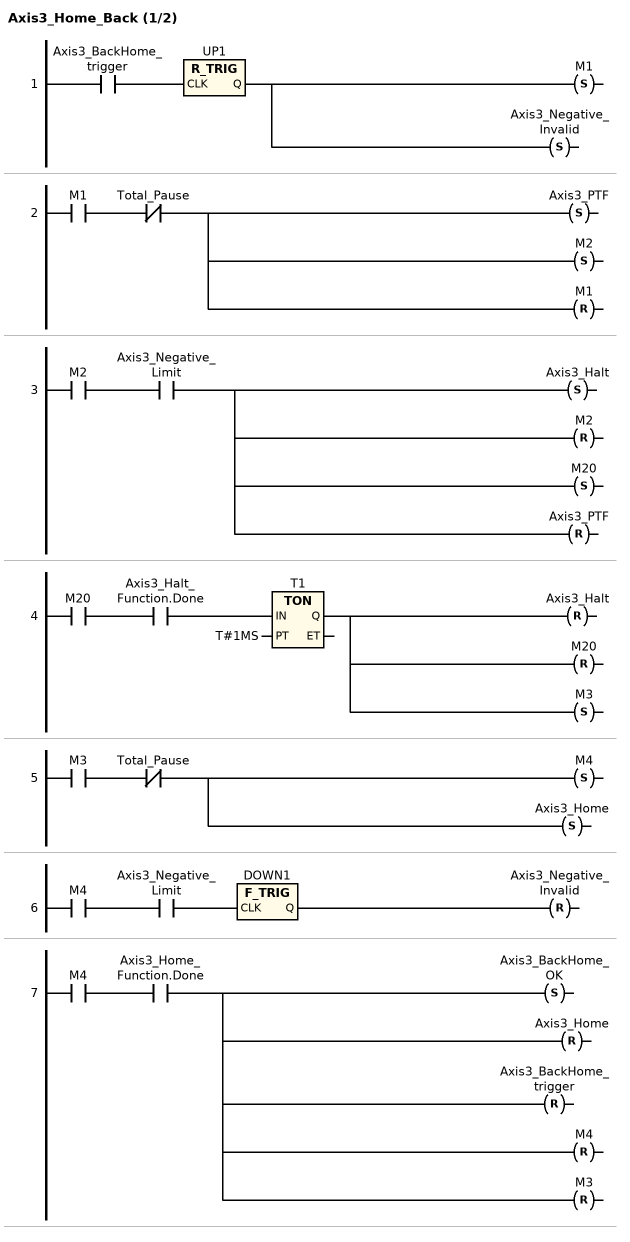
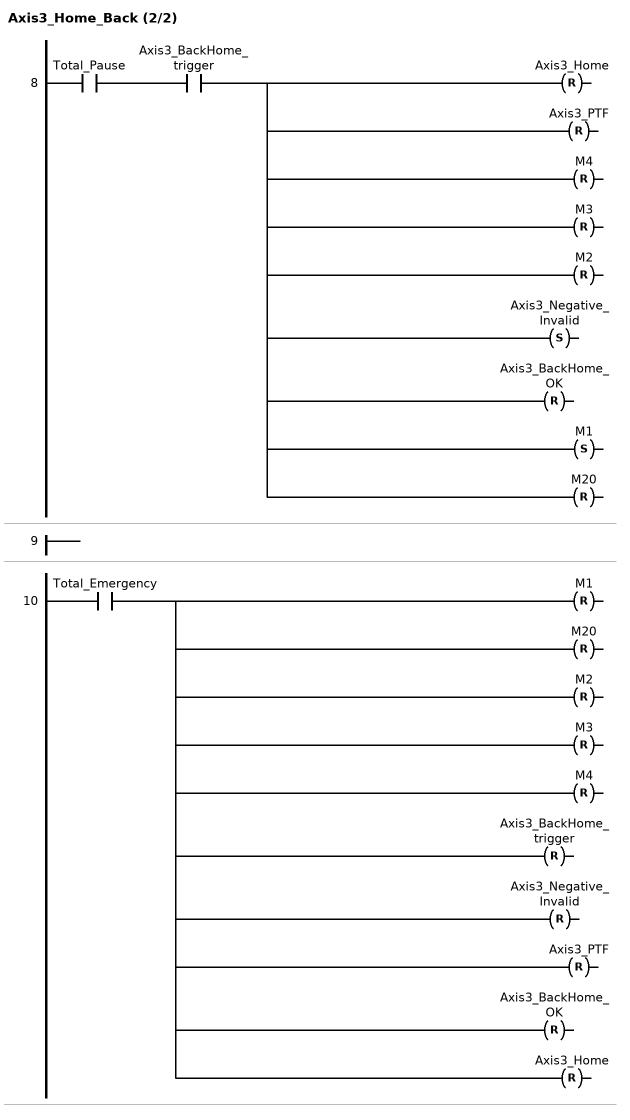
_LD_ (* Ladder Diagram *)
NETWORK 1
	[Axis3_BackHome_trigger] - UP1:R_TRIG(CLK: *) --- (S M1) (S Axis3_Negative_Invalid)
NETWORK 2
	[M1] - [/Total_Pause] --- (S Axis3_PTF) (S M2) (R M1)
NETWORK 3
	[M2] - [Axis3_Negative_Limit] --- (S Axis3_Halt) (R M2) (S M20) (R Axis3_PTF)
NETWORK 4
	[M20] - [Axis3_Halt_Function.Done] - T1:TON(IN: *, PT: T#1MS) --- (R Axis3_Halt) (R M20) (S M3)
NETWORK 5
	[M3] - [/Total_Pause] --- (S M4) (S Axis3_Home)
NETWORK 6
	[M4] - [Axis3_Negative_Limit] - DOWN1:F_TRIG(CLK: *) --- (R Axis3_Negative_Invalid)
NETWORK 7
	[M4] - [Axis3_Home_Function.Done] --- (S Axis3_BackHome_OK) (R Axis3_Home) (R Axis3_BackHome_trigger) (R M4) (R M3)
NETWORK 8
	[Total_Pause] - [Axis3_BackHome_trigger] --- (R Axis3_Home) (R Axis3_PTF) (R M4) (R M3) (R M2) (S Axis3_Negative_Invalid) (R Axis3_BackHome_OK) (S M1) (R M20)
NETWORK 9
	*
NETWORK 10
	[Total_Emergency] --- (R M1) (R M20) (R M2) (R M3) (R M4) (R Axis3_BackHome_trigger) (R Axis3_Negative_Invalid) (R Axis3_PTF) (R Axis3_BackHome_OK) (R Axis3_Home)
_END_LD_
(* the same logic as Structured Text *)
(* Network 1 *)
UP1(CLK := Axis3_BackHome_trigger);
IF UP1.Q THEN M1 := TRUE; Axis3_Negative_Invalid := TRUE; END_IF;
(* Network 2 *)
_p1 := M1 AND NOT Total_Pause;
IF _p1 THEN Axis3_PTF := TRUE; M2 := TRUE; M1 := FALSE; END_IF;
(* Network 3 *)
_p2 := M2 AND Axis3_Negative_Limit;
IF _p2 THEN Axis3_Halt := TRUE; M2 := FALSE; M20 := TRUE; Axis3_PTF := FALSE; END_IF;
(* Network 4 *)
T1(IN := M20 AND Axis3_Halt_Function.Done, PT := T#1MS);
IF T1.Q THEN Axis3_Halt := FALSE; M20 := FALSE; M3 := TRUE; END_IF;
(* Network 5 *)
IF M3 AND NOT Total_Pause THEN M4 := TRUE; Axis3_Home := TRUE; END_IF;
(* Network 6 *)
DOWN1(CLK := M4 AND Axis3_Negative_Limit);
IF DOWN1.Q THEN Axis3_Negative_Invalid := FALSE; END_IF;
(* Network 7 *)
_p3 := M4 AND Axis3_Home_Function.Done;
IF _p3 THEN Axis3_BackHome_OK := TRUE; Axis3_Home := FALSE; Axis3_BackHome_trigger := FALSE; M4 := FALSE; M3 := FALSE; END_IF;
(* Network 8 *)
IF Total_Pause AND Axis3_BackHome_trigger THEN Axis3_Home := FALSE; Axis3_PTF := FALSE; M4 := FALSE; M3 := FALSE; M2 := FALSE; Axis3_Negative_Invalid := TRUE; Axis3_BackHome_OK := FALSE; M1 := TRUE; M20 := FALSE; END_IF;
(* Network 9 *)
(* Network 10 *)
IF Total_Emergency THEN M1 := FALSE; M20 := FALSE; M2 := FALSE; M3 := FALSE; M4 := FALSE; Axis3_BackHome_trigger := FALSE; Axis3_Negative_Invalid := FALSE; Axis3_PTF := FALSE; Axis3_BackHome_OK := FALSE; Axis3_Home := FALSE; END_IF;
END_PROGRAM

(* POU Other_Folder/Home_Back/Axis4_Home_Back, LD *)
PROGRAM Axis4_Home_Back
VAR
	UP1: R_TRIG;
	M1: BOOL;
	M2: BOOL;
	UP2: R_TRIG;
	T1: TON;
	M3: BOOL;
	M4: BOOL;
	DOWN1: F_TRIG;
	M20: BOOL;
END_VAR
VAR (* helpers for the ST form of the networks *)
	_p1 : BOOL;
	_p2 : BOOL;
	_p3 : BOOL;
END_VAR
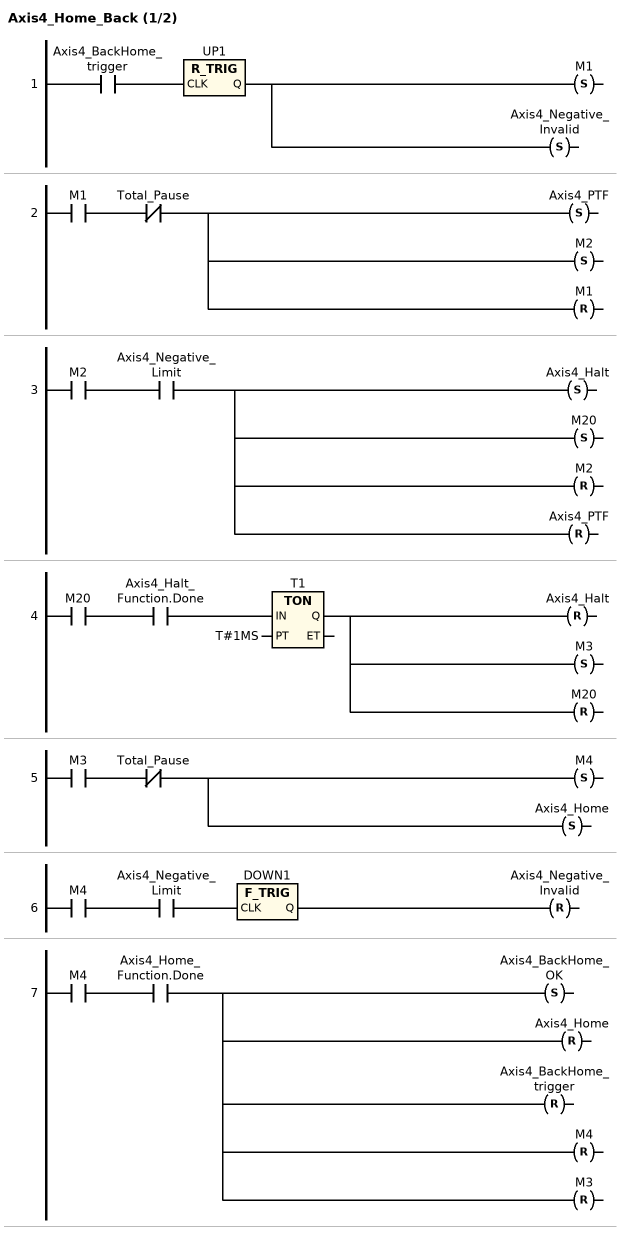
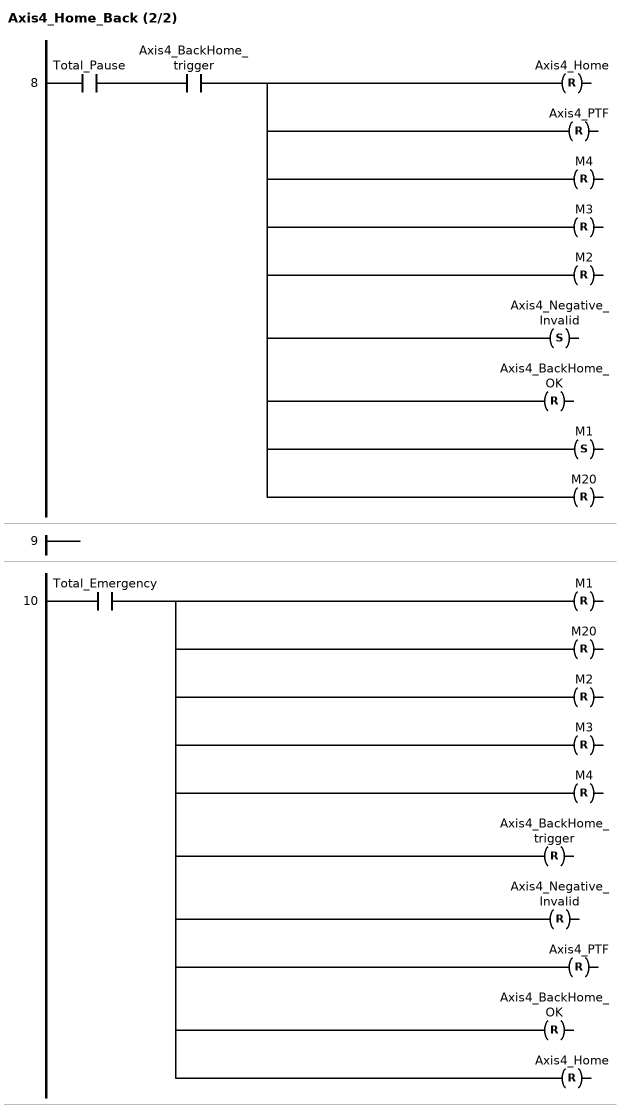
_LD_ (* Ladder Diagram *)
NETWORK 1
	[Axis4_BackHome_trigger] - UP1:R_TRIG(CLK: *) --- (S M1) (S Axis4_Negative_Invalid)
NETWORK 2
	[M1] - [/Total_Pause] --- (S Axis4_PTF) (S M2) (R M1)
NETWORK 3
	[M2] - [Axis4_Negative_Limit] --- (S Axis4_Halt) (S M20) (R M2) (R Axis4_PTF)
NETWORK 4
	[M20] - [Axis4_Halt_Function.Done] - T1:TON(IN: *, PT: T#1MS) --- (R Axis4_Halt) (S M3) (R M20)
NETWORK 5
	[M3] - [/Total_Pause] --- (S M4) (S Axis4_Home)
NETWORK 6
	[M4] - [Axis4_Negative_Limit] - DOWN1:F_TRIG(CLK: *) --- (R Axis4_Negative_Invalid)
NETWORK 7
	[M4] - [Axis4_Home_Function.Done] --- (S Axis4_BackHome_OK) (R Axis4_Home) (R Axis4_BackHome_trigger) (R M4) (R M3)
NETWORK 8
	[Total_Pause] - [Axis4_BackHome_trigger] --- (R Axis4_Home) (R Axis4_PTF) (R M4) (R M3) (R M2) (S Axis4_Negative_Invalid) (R Axis4_BackHome_OK) (S M1) (R M20)
NETWORK 9
	*
NETWORK 10
	[Total_Emergency] --- (R M1) (R M20) (R M2) (R M3) (R M4) (R Axis4_BackHome_trigger) (R Axis4_Negative_Invalid) (R Axis4_PTF) (R Axis4_BackHome_OK) (R Axis4_Home)
_END_LD_
(* the same logic as Structured Text *)
(* Network 1 *)
UP1(CLK := Axis4_BackHome_trigger);
IF UP1.Q THEN M1 := TRUE; Axis4_Negative_Invalid := TRUE; END_IF;
(* Network 2 *)
_p1 := M1 AND NOT Total_Pause;
IF _p1 THEN Axis4_PTF := TRUE; M2 := TRUE; M1 := FALSE; END_IF;
(* Network 3 *)
_p2 := M2 AND Axis4_Negative_Limit;
IF _p2 THEN Axis4_Halt := TRUE; M20 := TRUE; M2 := FALSE; Axis4_PTF := FALSE; END_IF;
(* Network 4 *)
T1(IN := M20 AND Axis4_Halt_Function.Done, PT := T#1MS);
IF T1.Q THEN Axis4_Halt := FALSE; M3 := TRUE; M20 := FALSE; END_IF;
(* Network 5 *)
IF M3 AND NOT Total_Pause THEN M4 := TRUE; Axis4_Home := TRUE; END_IF;
(* Network 6 *)
DOWN1(CLK := M4 AND Axis4_Negative_Limit);
IF DOWN1.Q THEN Axis4_Negative_Invalid := FALSE; END_IF;
(* Network 7 *)
_p3 := M4 AND Axis4_Home_Function.Done;
IF _p3 THEN Axis4_BackHome_OK := TRUE; Axis4_Home := FALSE; Axis4_BackHome_trigger := FALSE; M4 := FALSE; M3 := FALSE; END_IF;
(* Network 8 *)
IF Total_Pause AND Axis4_BackHome_trigger THEN Axis4_Home := FALSE; Axis4_PTF := FALSE; M4 := FALSE; M3 := FALSE; M2 := FALSE; Axis4_Negative_Invalid := TRUE; Axis4_BackHome_OK := FALSE; M1 := TRUE; M20 := FALSE; END_IF;
(* Network 9 *)
(* Network 10 *)
IF Total_Emergency THEN M1 := FALSE; M20 := FALSE; M2 := FALSE; M3 := FALSE; M4 := FALSE; Axis4_BackHome_trigger := FALSE; Axis4_Negative_Invalid := FALSE; Axis4_PTF := FALSE; Axis4_BackHome_OK := FALSE; Axis4_Home := FALSE; END_IF;
END_PROGRAM

(* POU Other_Folder/Home_Back/Axis5_Home_Back, LD *)
PROGRAM Axis5_Home_Back
VAR
	UP1: R_TRIG;
	M1: BOOL;
	M2: BOOL;
	UP2: R_TRIG;
	T1: TON;
	M3: BOOL;
	M4: BOOL;
	DOWN1: F_TRIG;
	M20: BOOL;
END_VAR
VAR (* helpers for the ST form of the networks *)
	_p1 : BOOL;
	_p2 : BOOL;
	_p3 : BOOL;
END_VAR
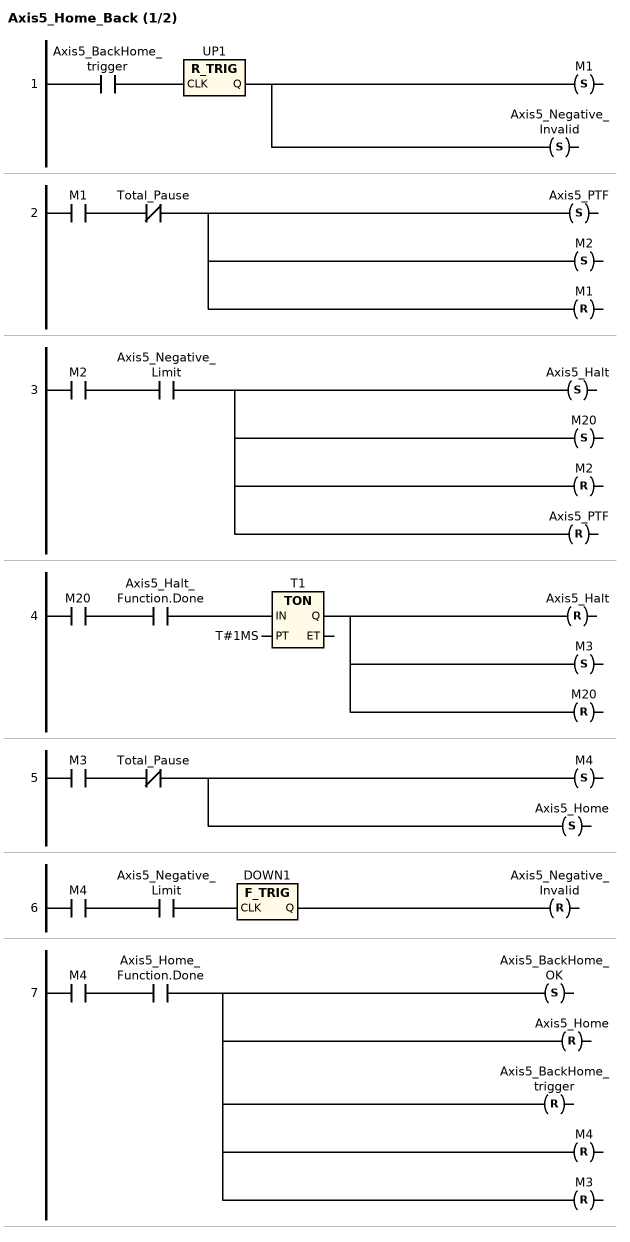
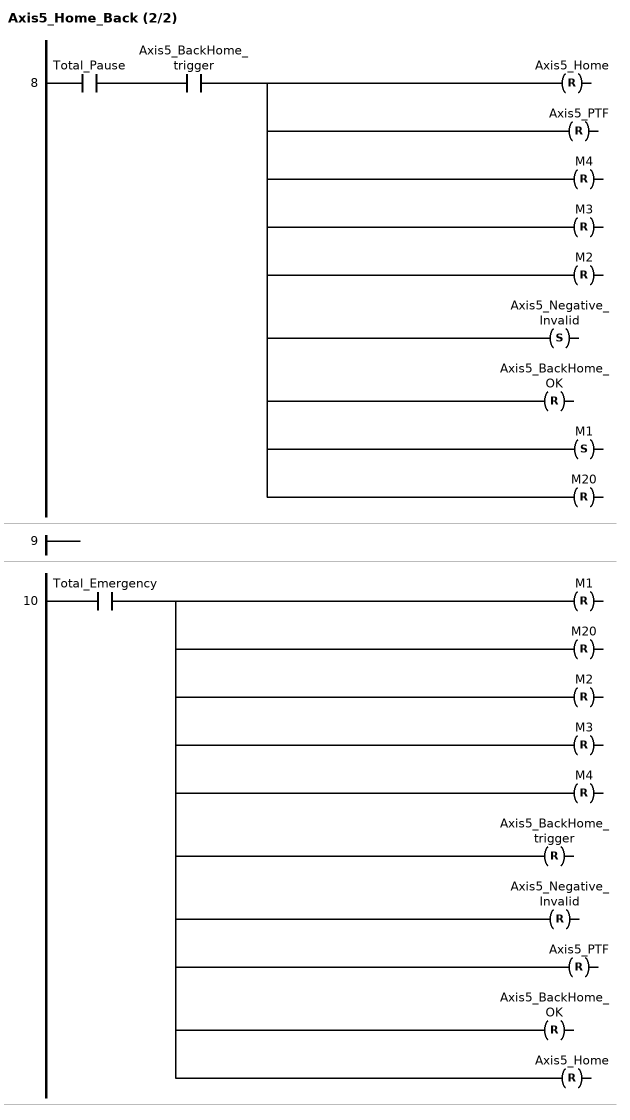
_LD_ (* Ladder Diagram *)
NETWORK 1
	[Axis5_BackHome_trigger] - UP1:R_TRIG(CLK: *) --- (S M1) (S Axis5_Negative_Invalid)
NETWORK 2
	[M1] - [/Total_Pause] --- (S Axis5_PTF) (S M2) (R M1)
NETWORK 3
	[M2] - [Axis5_Negative_Limit] --- (S Axis5_Halt) (S M20) (R M2) (R Axis5_PTF)
NETWORK 4
	[M20] - [Axis5_Halt_Function.Done] - T1:TON(IN: *, PT: T#1MS) --- (R Axis5_Halt) (S M3) (R M20)
NETWORK 5
	[M3] - [/Total_Pause] --- (S M4) (S Axis5_Home)
NETWORK 6
	[M4] - [Axis5_Negative_Limit] - DOWN1:F_TRIG(CLK: *) --- (R Axis5_Negative_Invalid)
NETWORK 7
	[M4] - [Axis5_Home_Function.Done] --- (S Axis5_BackHome_OK) (R Axis5_Home) (R Axis5_BackHome_trigger) (R M4) (R M3)
NETWORK 8
	[Total_Pause] - [Axis5_BackHome_trigger] --- (R Axis5_Home) (R Axis5_PTF) (R M4) (R M3) (R M2) (S Axis5_Negative_Invalid) (R Axis5_BackHome_OK) (S M1) (R M20)
NETWORK 9
	*
NETWORK 10
	[Total_Emergency] --- (R M1) (R M20) (R M2) (R M3) (R M4) (R Axis5_BackHome_trigger) (R Axis5_Negative_Invalid) (R Axis5_PTF) (R Axis5_BackHome_OK) (R Axis5_Home)
_END_LD_
(* the same logic as Structured Text *)
(* Network 1 *)
UP1(CLK := Axis5_BackHome_trigger);
IF UP1.Q THEN M1 := TRUE; Axis5_Negative_Invalid := TRUE; END_IF;
(* Network 2 *)
_p1 := M1 AND NOT Total_Pause;
IF _p1 THEN Axis5_PTF := TRUE; M2 := TRUE; M1 := FALSE; END_IF;
(* Network 3 *)
_p2 := M2 AND Axis5_Negative_Limit;
IF _p2 THEN Axis5_Halt := TRUE; M20 := TRUE; M2 := FALSE; Axis5_PTF := FALSE; END_IF;
(* Network 4 *)
T1(IN := M20 AND Axis5_Halt_Function.Done, PT := T#1MS);
IF T1.Q THEN Axis5_Halt := FALSE; M3 := TRUE; M20 := FALSE; END_IF;
(* Network 5 *)
IF M3 AND NOT Total_Pause THEN M4 := TRUE; Axis5_Home := TRUE; END_IF;
(* Network 6 *)
DOWN1(CLK := M4 AND Axis5_Negative_Limit);
IF DOWN1.Q THEN Axis5_Negative_Invalid := FALSE; END_IF;
(* Network 7 *)
_p3 := M4 AND Axis5_Home_Function.Done;
IF _p3 THEN Axis5_BackHome_OK := TRUE; Axis5_Home := FALSE; Axis5_BackHome_trigger := FALSE; M4 := FALSE; M3 := FALSE; END_IF;
(* Network 8 *)
IF Total_Pause AND Axis5_BackHome_trigger THEN Axis5_Home := FALSE; Axis5_PTF := FALSE; M4 := FALSE; M3 := FALSE; M2 := FALSE; Axis5_Negative_Invalid := TRUE; Axis5_BackHome_OK := FALSE; M1 := TRUE; M20 := FALSE; END_IF;
(* Network 9 *)
(* Network 10 *)
IF Total_Emergency THEN M1 := FALSE; M20 := FALSE; M2 := FALSE; M3 := FALSE; M4 := FALSE; Axis5_BackHome_trigger := FALSE; Axis5_Negative_Invalid := FALSE; Axis5_PTF := FALSE; Axis5_BackHome_OK := FALSE; Axis5_Home := FALSE; END_IF;
END_PROGRAM

(* POU Other_Folder/Home_Back/Axis6_Home_Back, LD *)
PROGRAM Axis6_Home_Back
VAR
	UP1: R_TRIG;
	M1: BOOL;
	M2: BOOL;
	UP2: R_TRIG;
	T1: TON;
	M3: BOOL;
	M4: BOOL;
	DOWN1: F_TRIG;
	M20: BOOL;
END_VAR
VAR (* helpers for the ST form of the networks *)
	_p1 : BOOL;
	_p2 : BOOL;
	_p3 : BOOL;
END_VAR
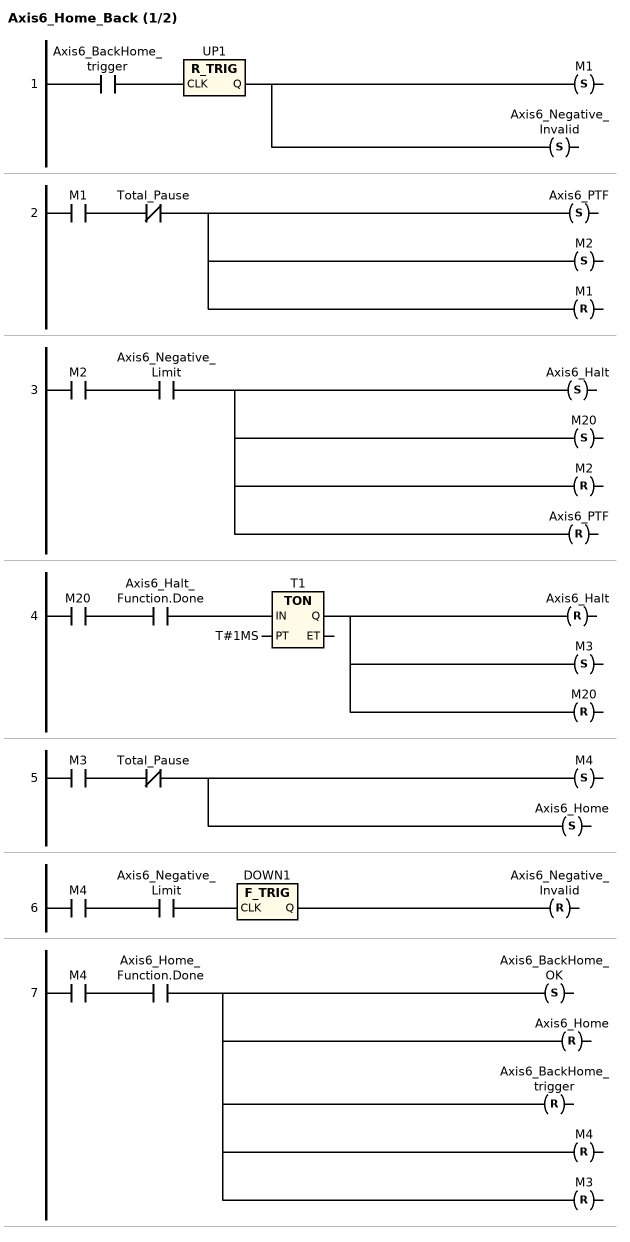
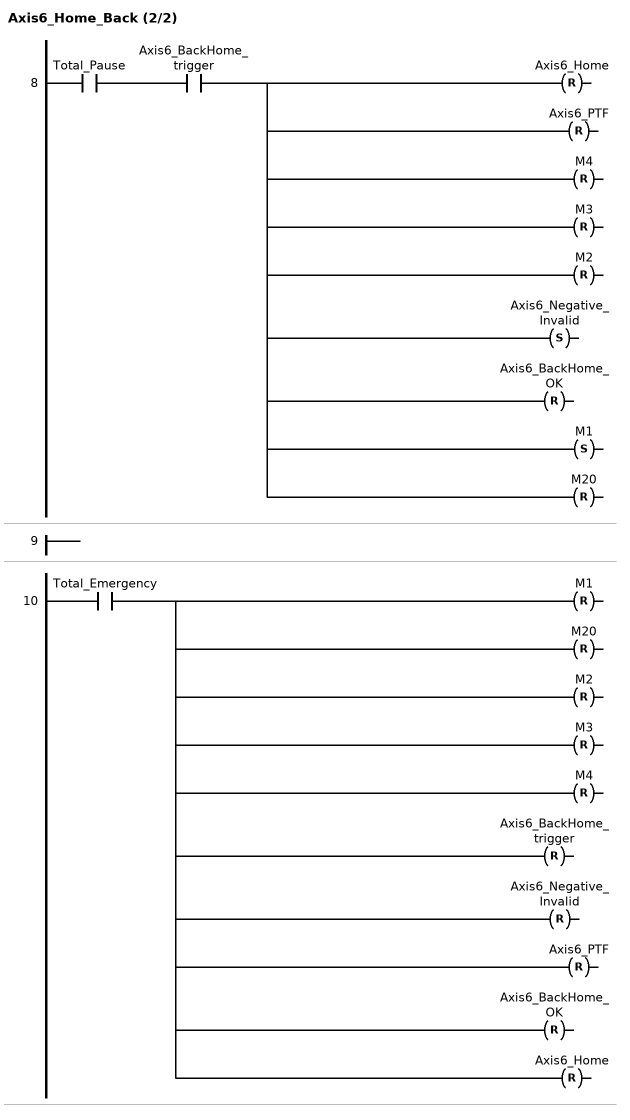
_LD_ (* Ladder Diagram *)
NETWORK 1
	[Axis6_BackHome_trigger] - UP1:R_TRIG(CLK: *) --- (S M1) (S Axis6_Negative_Invalid)
NETWORK 2
	[M1] - [/Total_Pause] --- (S Axis6_PTF) (S M2) (R M1)
NETWORK 3
	[M2] - [Axis6_Negative_Limit] --- (S Axis6_Halt) (S M20) (R M2) (R Axis6_PTF)
NETWORK 4
	[M20] - [Axis6_Halt_Function.Done] - T1:TON(IN: *, PT: T#1MS) --- (R Axis6_Halt) (S M3) (R M20)
NETWORK 5
	[M3] - [/Total_Pause] --- (S M4) (S Axis6_Home)
NETWORK 6
	[M4] - [Axis6_Negative_Limit] - DOWN1:F_TRIG(CLK: *) --- (R Axis6_Negative_Invalid)
NETWORK 7
	[M4] - [Axis6_Home_Function.Done] --- (S Axis6_BackHome_OK) (R Axis6_Home) (R Axis6_BackHome_trigger) (R M4) (R M3)
NETWORK 8
	[Total_Pause] - [Axis6_BackHome_trigger] --- (R Axis6_Home) (R Axis6_PTF) (R M4) (R M3) (R M2) (S Axis6_Negative_Invalid) (R Axis6_BackHome_OK) (S M1) (R M20)
NETWORK 9
	*
NETWORK 10
	[Total_Emergency] --- (R M1) (R M20) (R M2) (R M3) (R M4) (R Axis6_BackHome_trigger) (R Axis6_Negative_Invalid) (R Axis6_PTF) (R Axis6_BackHome_OK) (R Axis6_Home)
_END_LD_
(* the same logic as Structured Text *)
(* Network 1 *)
UP1(CLK := Axis6_BackHome_trigger);
IF UP1.Q THEN M1 := TRUE; Axis6_Negative_Invalid := TRUE; END_IF;
(* Network 2 *)
_p1 := M1 AND NOT Total_Pause;
IF _p1 THEN Axis6_PTF := TRUE; M2 := TRUE; M1 := FALSE; END_IF;
(* Network 3 *)
_p2 := M2 AND Axis6_Negative_Limit;
IF _p2 THEN Axis6_Halt := TRUE; M20 := TRUE; M2 := FALSE; Axis6_PTF := FALSE; END_IF;
(* Network 4 *)
T1(IN := M20 AND Axis6_Halt_Function.Done, PT := T#1MS);
IF T1.Q THEN Axis6_Halt := FALSE; M3 := TRUE; M20 := FALSE; END_IF;
(* Network 5 *)
IF M3 AND NOT Total_Pause THEN M4 := TRUE; Axis6_Home := TRUE; END_IF;
(* Network 6 *)
DOWN1(CLK := M4 AND Axis6_Negative_Limit);
IF DOWN1.Q THEN Axis6_Negative_Invalid := FALSE; END_IF;
(* Network 7 *)
_p3 := M4 AND Axis6_Home_Function.Done;
IF _p3 THEN Axis6_BackHome_OK := TRUE; Axis6_Home := FALSE; Axis6_BackHome_trigger := FALSE; M4 := FALSE; M3 := FALSE; END_IF;
(* Network 8 *)
IF Total_Pause AND Axis6_BackHome_trigger THEN Axis6_Home := FALSE; Axis6_PTF := FALSE; M4 := FALSE; M3 := FALSE; M2 := FALSE; Axis6_Negative_Invalid := TRUE; Axis6_BackHome_OK := FALSE; M1 := TRUE; M20 := FALSE; END_IF;
(* Network 9 *)
(* Network 10 *)
IF Total_Emergency THEN M1 := FALSE; M20 := FALSE; M2 := FALSE; M3 := FALSE; M4 := FALSE; Axis6_BackHome_trigger := FALSE; Axis6_Negative_Invalid := FALSE; Axis6_PTF := FALSE; Axis6_BackHome_OK := FALSE; Axis6_Home := FALSE; END_IF;
END_PROGRAM

(* POU Other_Folder/Home_Back/Axis7_Home_Back, LD *)
PROGRAM Axis7_Home_Back
VAR
	UP1: R_TRIG;
	M1: BOOL;
	M2: BOOL;
	UP2: R_TRIG;
	T1: TON;
	M3: BOOL;
	M4: BOOL;
	DOWN1: F_TRIG;
	M20: BOOL;
END_VAR
VAR (* helpers for the ST form of the networks *)
	_p1 : BOOL;
	_p2 : BOOL;
	_p3 : BOOL;
END_VAR
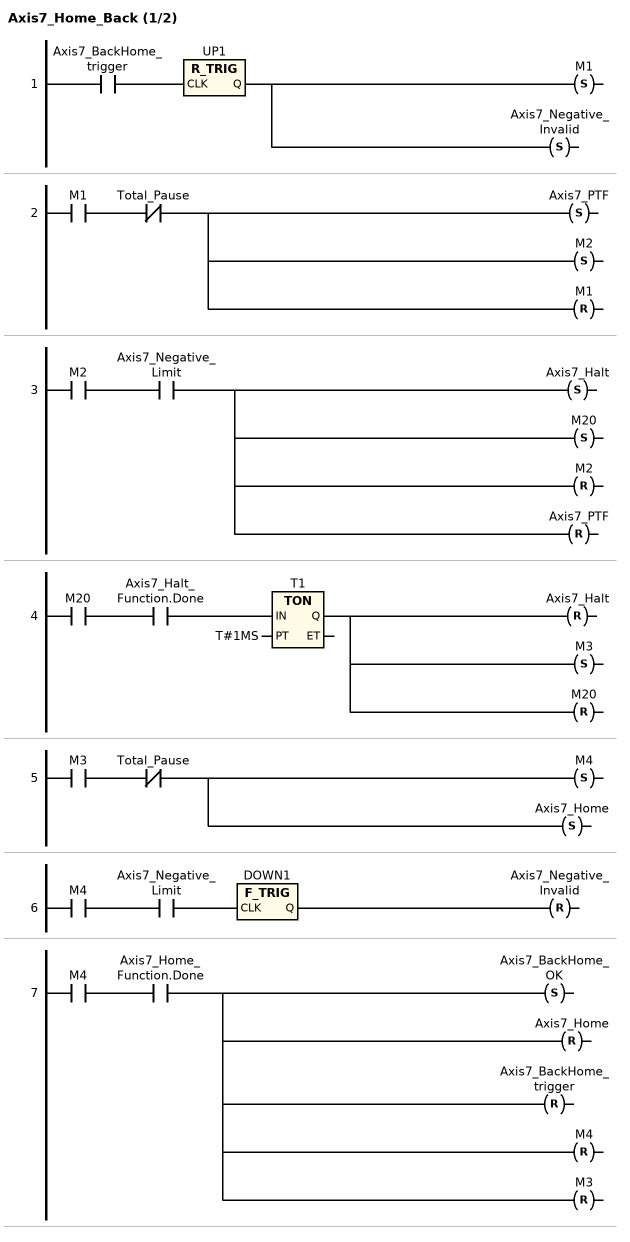
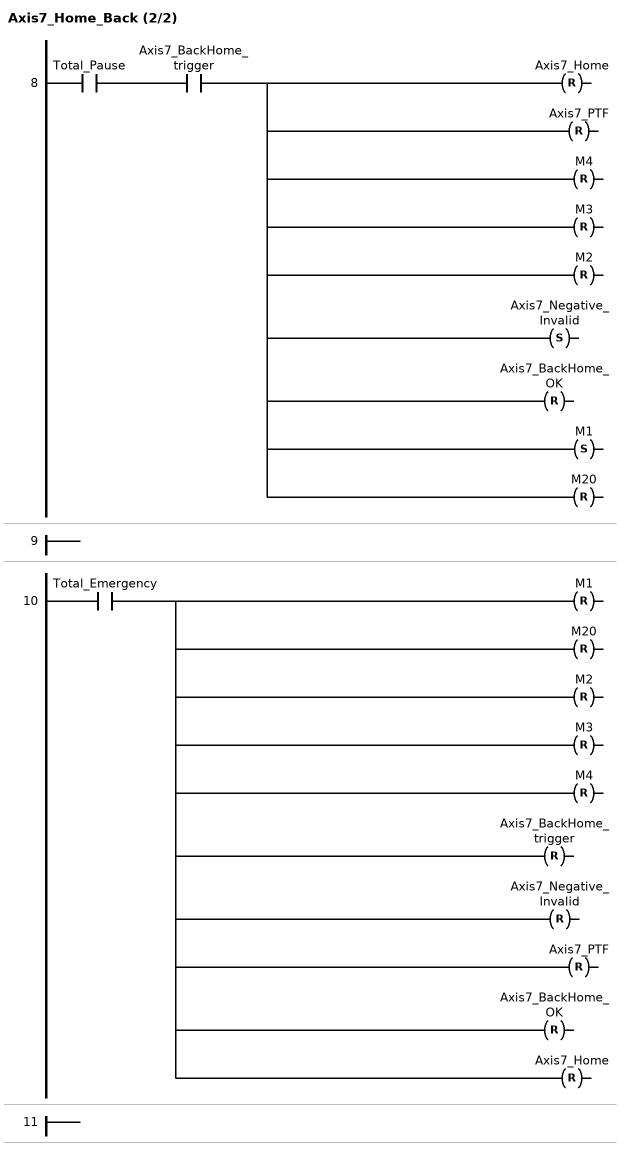
_LD_ (* Ladder Diagram *)
NETWORK 1
	[Axis7_BackHome_trigger] - UP1:R_TRIG(CLK: *) --- (S M1) (S Axis7_Negative_Invalid)
NETWORK 2
	[M1] - [/Total_Pause] --- (S Axis7_PTF) (S M2) (R M1)
NETWORK 3
	[M2] - [Axis7_Negative_Limit] --- (S Axis7_Halt) (S M20) (R M2) (R Axis7_PTF)
NETWORK 4
	[M20] - [Axis7_Halt_Function.Done] - T1:TON(IN: *, PT: T#1MS) --- (R Axis7_Halt) (S M3) (R M20)
NETWORK 5
	[M3] - [/Total_Pause] --- (S M4) (S Axis7_Home)
NETWORK 6
	[M4] - [Axis7_Negative_Limit] - DOWN1:F_TRIG(CLK: *) --- (R Axis7_Negative_Invalid)
NETWORK 7
	[M4] - [Axis7_Home_Function.Done] --- (S Axis7_BackHome_OK) (R Axis7_Home) (R Axis7_BackHome_trigger) (R M4) (R M3)
NETWORK 8
	[Total_Pause] - [Axis7_BackHome_trigger] --- (R Axis7_Home) (R Axis7_PTF) (R M4) (R M3) (R M2) (S Axis7_Negative_Invalid) (R Axis7_BackHome_OK) (S M1) (R M20)
NETWORK 9
	*
NETWORK 10
	[Total_Emergency] --- (R M1) (R M20) (R M2) (R M3) (R M4) (R Axis7_BackHome_trigger) (R Axis7_Negative_Invalid) (R Axis7_PTF) (R Axis7_BackHome_OK) (R Axis7_Home)
NETWORK 11
	*
_END_LD_
(* the same logic as Structured Text *)
(* Network 1 *)
UP1(CLK := Axis7_BackHome_trigger);
IF UP1.Q THEN M1 := TRUE; Axis7_Negative_Invalid := TRUE; END_IF;
(* Network 2 *)
_p1 := M1 AND NOT Total_Pause;
IF _p1 THEN Axis7_PTF := TRUE; M2 := TRUE; M1 := FALSE; END_IF;
(* Network 3 *)
_p2 := M2 AND Axis7_Negative_Limit;
IF _p2 THEN Axis7_Halt := TRUE; M20 := TRUE; M2 := FALSE; Axis7_PTF := FALSE; END_IF;
(* Network 4 *)
T1(IN := M20 AND Axis7_Halt_Function.Done, PT := T#1MS);
IF T1.Q THEN Axis7_Halt := FALSE; M3 := TRUE; M20 := FALSE; END_IF;
(* Network 5 *)
IF M3 AND NOT Total_Pause THEN M4 := TRUE; Axis7_Home := TRUE; END_IF;
(* Network 6 *)
DOWN1(CLK := M4 AND Axis7_Negative_Limit);
IF DOWN1.Q THEN Axis7_Negative_Invalid := FALSE; END_IF;
(* Network 7 *)
_p3 := M4 AND Axis7_Home_Function.Done;
IF _p3 THEN Axis7_BackHome_OK := TRUE; Axis7_Home := FALSE; Axis7_BackHome_trigger := FALSE; M4 := FALSE; M3 := FALSE; END_IF;
(* Network 8 *)
IF Total_Pause AND Axis7_BackHome_trigger THEN Axis7_Home := FALSE; Axis7_PTF := FALSE; M4 := FALSE; M3 := FALSE; M2 := FALSE; Axis7_Negative_Invalid := TRUE; Axis7_BackHome_OK := FALSE; M1 := TRUE; M20 := FALSE; END_IF;
(* Network 9 *)
(* Network 10 *)
IF Total_Emergency THEN M1 := FALSE; M20 := FALSE; M2 := FALSE; M3 := FALSE; M4 := FALSE; Axis7_BackHome_trigger := FALSE; Axis7_Negative_Invalid := FALSE; Axis7_PTF := FALSE; Axis7_BackHome_OK := FALSE; Axis7_Home := FALSE; END_IF;
(* Network 11 *)
END_PROGRAM

(* POU Other_Folder/Home_Back/Axis8_Home_Back, LD *)
PROGRAM Axis8_Home_Back
VAR
	UP1: R_TRIG;
	M1: BOOL;
	M2: BOOL;
	UP2: R_TRIG;
	T1: TON;
	M3: BOOL;
	M4: BOOL;
	DOWN1: F_TRIG;
	M20: BOOL;
END_VAR
VAR (* helpers for the ST form of the networks *)
	_p1 : BOOL;
	_p2 : BOOL;
	_p3 : BOOL;
END_VAR
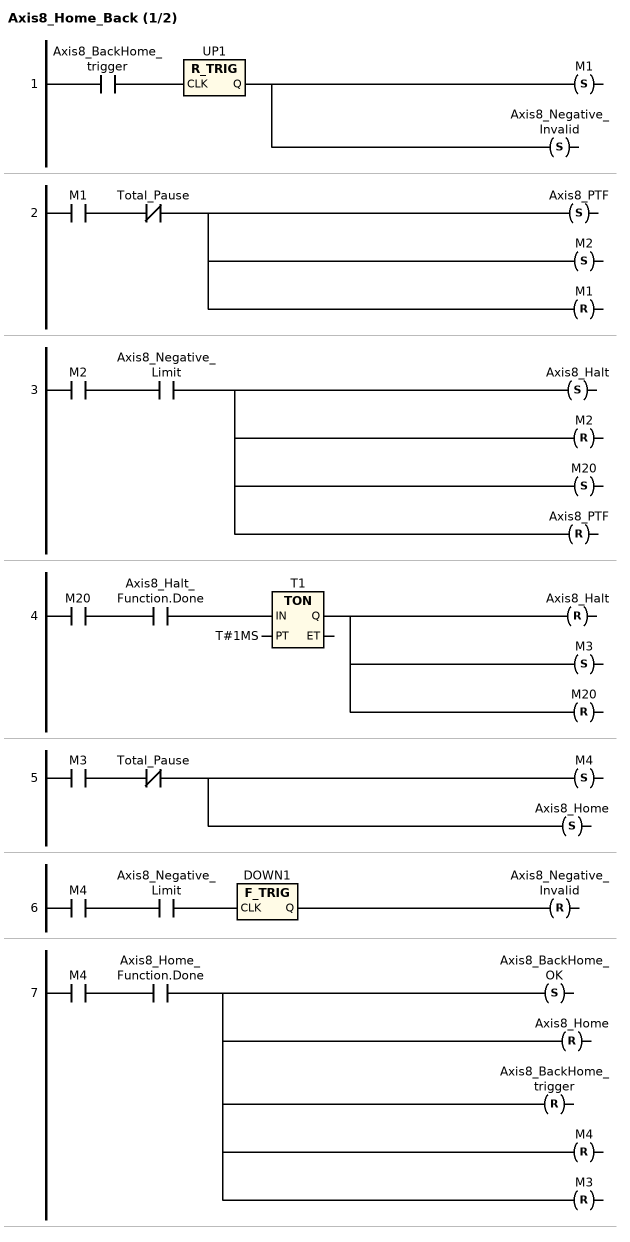
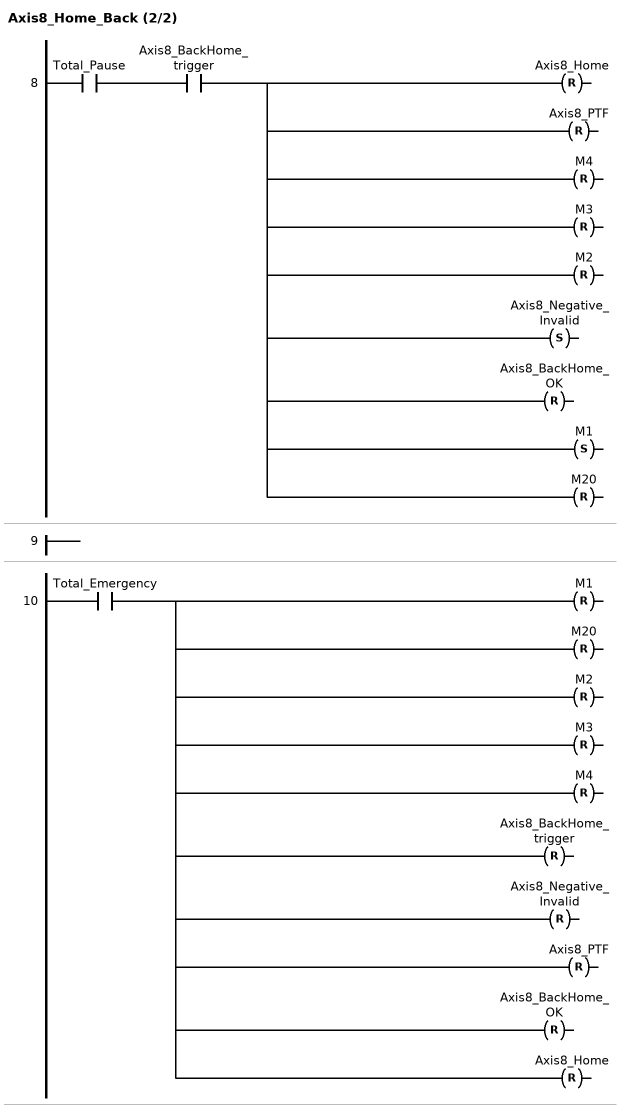
_LD_ (* Ladder Diagram *)
NETWORK 1
	[Axis8_BackHome_trigger] - UP1:R_TRIG(CLK: *) --- (S M1) (S Axis8_Negative_Invalid)
NETWORK 2
	[M1] - [/Total_Pause] --- (S Axis8_PTF) (S M2) (R M1)
NETWORK 3
	[M2] - [Axis8_Negative_Limit] --- (S Axis8_Halt) (R M2) (S M20) (R Axis8_PTF)
NETWORK 4
	[M20] - [Axis8_Halt_Function.Done] - T1:TON(IN: *, PT: T#1MS) --- (R Axis8_Halt) (S M3) (R M20)
NETWORK 5
	[M3] - [/Total_Pause] --- (S M4) (S Axis8_Home)
NETWORK 6
	[M4] - [Axis8_Negative_Limit] - DOWN1:F_TRIG(CLK: *) --- (R Axis8_Negative_Invalid)
NETWORK 7
	[M4] - [Axis8_Home_Function.Done] --- (S Axis8_BackHome_OK) (R Axis8_Home) (R Axis8_BackHome_trigger) (R M4) (R M3)
NETWORK 8
	[Total_Pause] - [Axis8_BackHome_trigger] --- (R Axis8_Home) (R Axis8_PTF) (R M4) (R M3) (R M2) (S Axis8_Negative_Invalid) (R Axis8_BackHome_OK) (S M1) (R M20)
NETWORK 9
	*
NETWORK 10
	[Total_Emergency] --- (R M1) (R M20) (R M2) (R M3) (R M4) (R Axis8_BackHome_trigger) (R Axis8_Negative_Invalid) (R Axis8_PTF) (R Axis8_BackHome_OK) (R Axis8_Home)
_END_LD_
(* the same logic as Structured Text *)
(* Network 1 *)
UP1(CLK := Axis8_BackHome_trigger);
IF UP1.Q THEN M1 := TRUE; Axis8_Negative_Invalid := TRUE; END_IF;
(* Network 2 *)
_p1 := M1 AND NOT Total_Pause;
IF _p1 THEN Axis8_PTF := TRUE; M2 := TRUE; M1 := FALSE; END_IF;
(* Network 3 *)
_p2 := M2 AND Axis8_Negative_Limit;
IF _p2 THEN Axis8_Halt := TRUE; M2 := FALSE; M20 := TRUE; Axis8_PTF := FALSE; END_IF;
(* Network 4 *)
T1(IN := M20 AND Axis8_Halt_Function.Done, PT := T#1MS);
IF T1.Q THEN Axis8_Halt := FALSE; M3 := TRUE; M20 := FALSE; END_IF;
(* Network 5 *)
IF M3 AND NOT Total_Pause THEN M4 := TRUE; Axis8_Home := TRUE; END_IF;
(* Network 6 *)
DOWN1(CLK := M4 AND Axis8_Negative_Limit);
IF DOWN1.Q THEN Axis8_Negative_Invalid := FALSE; END_IF;
(* Network 7 *)
_p3 := M4 AND Axis8_Home_Function.Done;
IF _p3 THEN Axis8_BackHome_OK := TRUE; Axis8_Home := FALSE; Axis8_BackHome_trigger := FALSE; M4 := FALSE; M3 := FALSE; END_IF;
(* Network 8 *)
IF Total_Pause AND Axis8_BackHome_trigger THEN Axis8_Home := FALSE; Axis8_PTF := FALSE; M4 := FALSE; M3 := FALSE; M2 := FALSE; Axis8_Negative_Invalid := TRUE; Axis8_BackHome_OK := FALSE; M1 := TRUE; M20 := FALSE; END_IF;
(* Network 9 *)
(* Network 10 *)
IF Total_Emergency THEN M1 := FALSE; M20 := FALSE; M2 := FALSE; M3 := FALSE; M4 := FALSE; Axis8_BackHome_trigger := FALSE; Axis8_Negative_Invalid := FALSE; Axis8_PTF := FALSE; Axis8_BackHome_OK := FALSE; Axis8_Home := FALSE; END_IF;
END_PROGRAM

(* POU Other_Folder/Home_Back/Axis9_Home_Back, LD *)
PROGRAM Axis9_Home_Back
VAR
	UP1: R_TRIG;
	M1: BOOL;
	M2: BOOL;
	UP2: R_TRIG;
	T1: TON;
	M3: BOOL;
	M4: BOOL;
	DOWN1: F_TRIG;
	M20: BOOL;
END_VAR
VAR (* helpers for the ST form of the networks *)
	_p1 : BOOL;
	_p2 : BOOL;
	_p3 : BOOL;
END_VAR
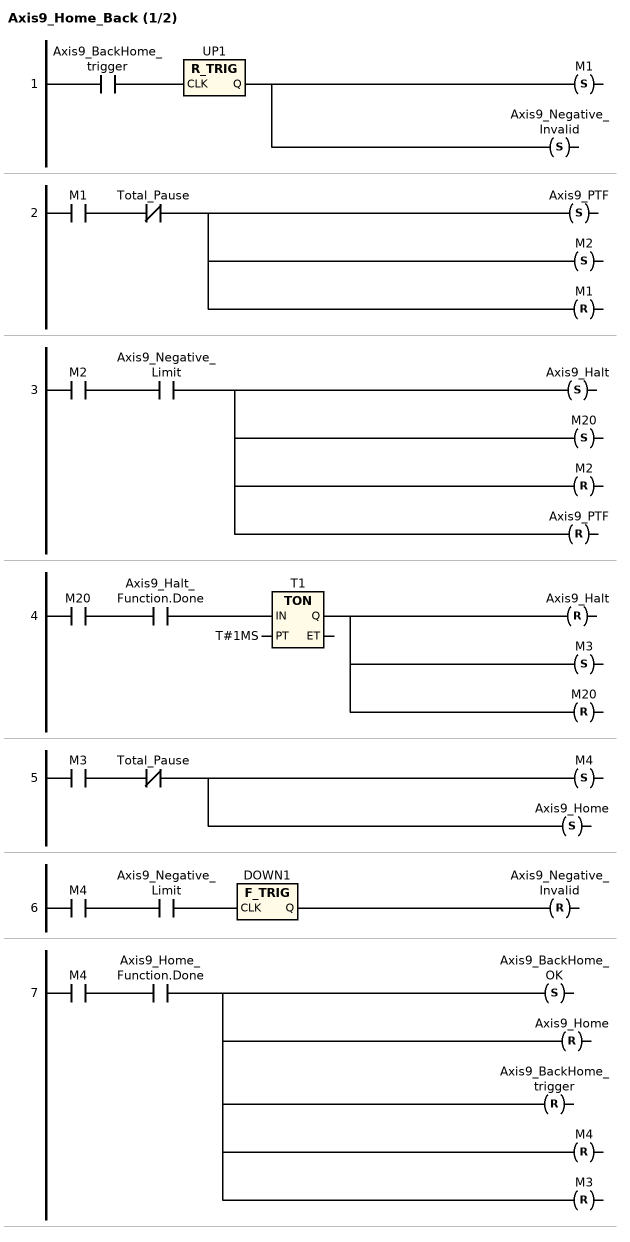
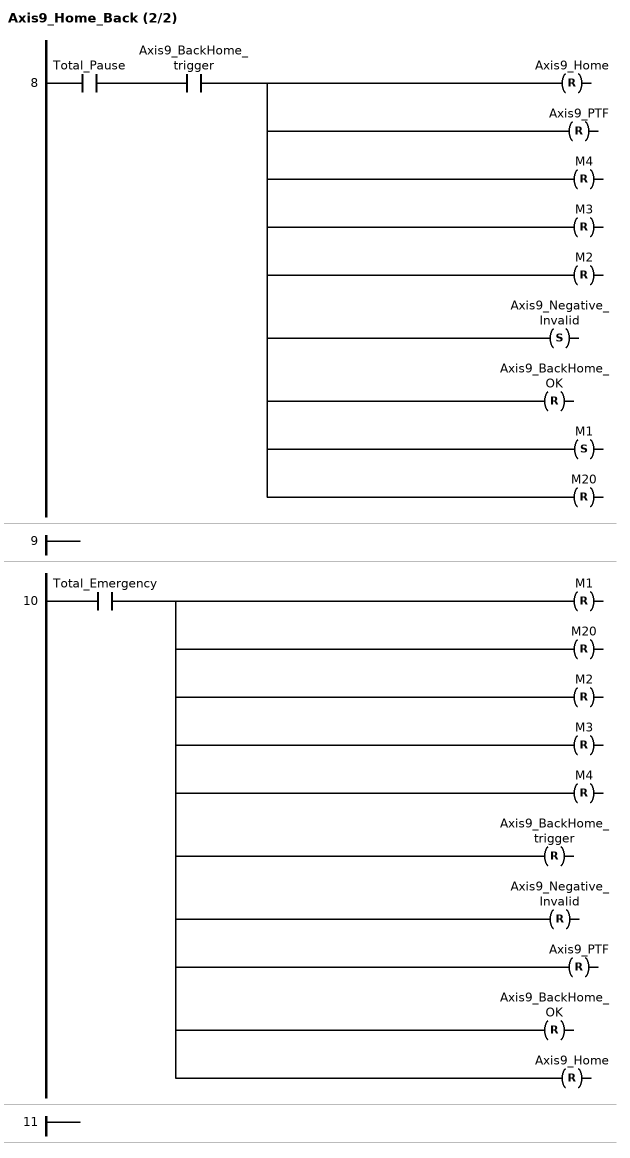
_LD_ (* Ladder Diagram *)
NETWORK 1
	[Axis9_BackHome_trigger] - UP1:R_TRIG(CLK: *) --- (S M1) (S Axis9_Negative_Invalid)
NETWORK 2
	[M1] - [/Total_Pause] --- (S Axis9_PTF) (S M2) (R M1)
NETWORK 3
	[M2] - [Axis9_Negative_Limit] --- (S Axis9_Halt) (S M20) (R M2) (R Axis9_PTF)
NETWORK 4
	[M20] - [Axis9_Halt_Function.Done] - T1:TON(IN: *, PT: T#1MS) --- (R Axis9_Halt) (S M3) (R M20)
NETWORK 5
	[M3] - [/Total_Pause] --- (S M4) (S Axis9_Home)
NETWORK 6
	[M4] - [Axis9_Negative_Limit] - DOWN1:F_TRIG(CLK: *) --- (R Axis9_Negative_Invalid)
NETWORK 7
	[M4] - [Axis9_Home_Function.Done] --- (S Axis9_BackHome_OK) (R Axis9_Home) (R Axis9_BackHome_trigger) (R M4) (R M3)
NETWORK 8
	[Total_Pause] - [Axis9_BackHome_trigger] --- (R Axis9_Home) (R Axis9_PTF) (R M4) (R M3) (R M2) (S Axis9_Negative_Invalid) (R Axis9_BackHome_OK) (S M1) (R M20)
NETWORK 9
	*
NETWORK 10
	[Total_Emergency] --- (R M1) (R M20) (R M2) (R M3) (R M4) (R Axis9_BackHome_trigger) (R Axis9_Negative_Invalid) (R Axis9_PTF) (R Axis9_BackHome_OK) (R Axis9_Home)
NETWORK 11
	*
_END_LD_
(* the same logic as Structured Text *)
(* Network 1 *)
UP1(CLK := Axis9_BackHome_trigger);
IF UP1.Q THEN M1 := TRUE; Axis9_Negative_Invalid := TRUE; END_IF;
(* Network 2 *)
_p1 := M1 AND NOT Total_Pause;
IF _p1 THEN Axis9_PTF := TRUE; M2 := TRUE; M1 := FALSE; END_IF;
(* Network 3 *)
_p2 := M2 AND Axis9_Negative_Limit;
IF _p2 THEN Axis9_Halt := TRUE; M20 := TRUE; M2 := FALSE; Axis9_PTF := FALSE; END_IF;
(* Network 4 *)
T1(IN := M20 AND Axis9_Halt_Function.Done, PT := T#1MS);
IF T1.Q THEN Axis9_Halt := FALSE; M3 := TRUE; M20 := FALSE; END_IF;
(* Network 5 *)
IF M3 AND NOT Total_Pause THEN M4 := TRUE; Axis9_Home := TRUE; END_IF;
(* Network 6 *)
DOWN1(CLK := M4 AND Axis9_Negative_Limit);
IF DOWN1.Q THEN Axis9_Negative_Invalid := FALSE; END_IF;
(* Network 7 *)
_p3 := M4 AND Axis9_Home_Function.Done;
IF _p3 THEN Axis9_BackHome_OK := TRUE; Axis9_Home := FALSE; Axis9_BackHome_trigger := FALSE; M4 := FALSE; M3 := FALSE; END_IF;
(* Network 8 *)
IF Total_Pause AND Axis9_BackHome_trigger THEN Axis9_Home := FALSE; Axis9_PTF := FALSE; M4 := FALSE; M3 := FALSE; M2 := FALSE; Axis9_Negative_Invalid := TRUE; Axis9_BackHome_OK := FALSE; M1 := TRUE; M20 := FALSE; END_IF;
(* Network 9 *)
(* Network 10 *)
IF Total_Emergency THEN M1 := FALSE; M20 := FALSE; M2 := FALSE; M3 := FALSE; M4 := FALSE; Axis9_BackHome_trigger := FALSE; Axis9_Negative_Invalid := FALSE; Axis9_PTF := FALSE; Axis9_BackHome_OK := FALSE; Axis9_Home := FALSE; END_IF;
(* Network 11 *)
END_PROGRAM

(* POU Other_Folder/Home_Back/Axis10_Home_Back, LD *)
PROGRAM Axis10_Home_Back
VAR
	UP1: R_TRIG;
	M1: BOOL;
	M2: BOOL;
	UP2: R_TRIG;
	T1: TON;
	M3: BOOL;
	M4: BOOL;
	DOWN1: F_TRIG;
	M20: BOOL;
END_VAR
VAR (* helpers for the ST form of the networks *)
	_p1 : BOOL;
	_p2 : BOOL;
	_p3 : BOOL;
END_VAR
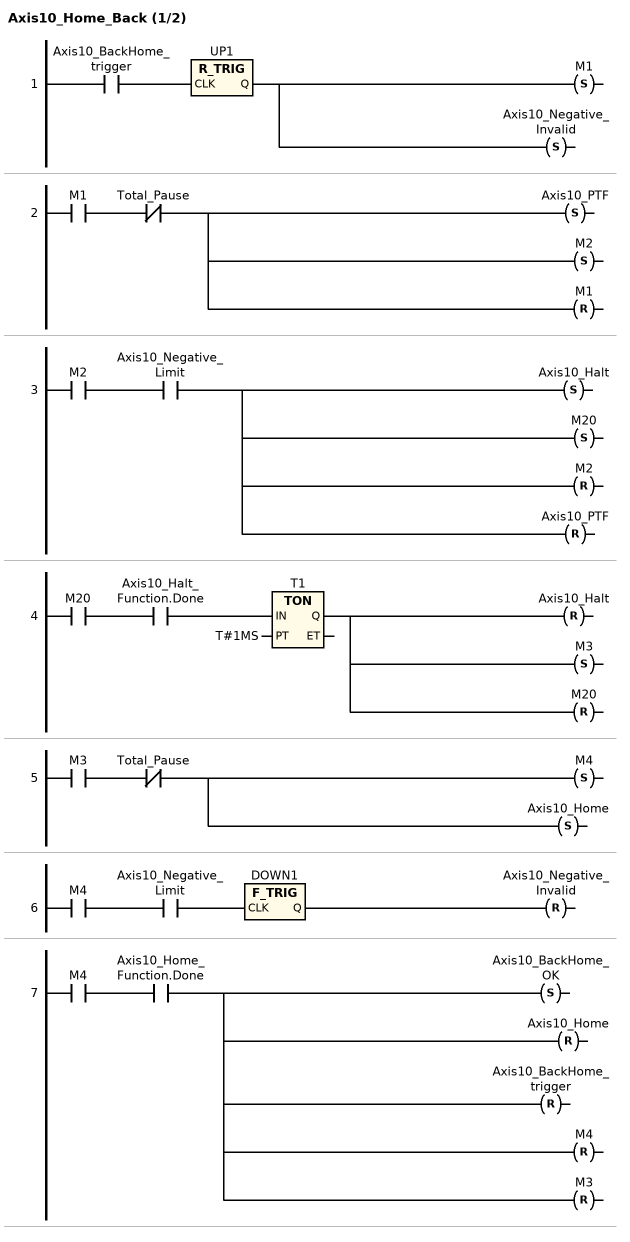
